(* IEC 61131-3 sources: Dev/Dev_V200/200 (part 10) *)

      iov : ARRAY[0.._Nh_CFG] OF FILT_LIST := [    // v hlavicke je RIADOK a v STLPCOCH su DEV, ktore ho mozu spustat (budu v prowse pre vyber)
            (),     	//  0 Empty
            (),    	//  1 Rmpty Rom
            (),    	//  2 Empty Cat
            (),    	//  3 Empty Zon
//                 0         5         10        15        20        25        30        35	      40        45	     50        55	       60        65
            (n := [0,0,0,0,0,0,0,0,0,0,0,0,0,1,1,1,0,0,0,0,0,0,0,0,0,0,0,0,0,0,0,0,0,0,0,0,0,0,0,0,1,0,0,0,0,0,0,0,0,0,1,0,0,0,0,0,0,0,0,0,0,0,0,0,0,0]) ,    //  4 scn  sceny
            (n := [0,0,0,0,0,0,0,0,0,0,0,0,0,1,1,1,0,0,0,0,0,0,0,0,1,0,0,0,0,0,0,0,0,0,0,0,0,0,0,0,1,0,0,0,0,0,0,0,0,0,1,0,0,0,0,0,0,0,0,0,0,0,0,0,0,0]) ,    //  5 act  akcie
            (n := [0,0,0,0,0,0,0,0,0,0,1,1,1,1,1,0,0,0,0,0,0,0,0,0,0,0,0,0,0,0,0,0,0,0,0,0,0,0,0,0,1,0,0,1,1,0,0,0,0,0,0,0,0,0,0,0,0,0,0,0,0,0,0,0,0,0]) ,    //  6 het  modul kurenia
            (n := [0,0,0,0,0,0,0,0,0,0,0,0,0,0,0,0,0,0,0,0,0,0,0,0,0,0,0,0,0,0,0,0,0,0,0,0,0,0,0,0,0,0,0,0,0,0,0,0,0,0,0,0,0,0,0,0,0,0,0,0,0,0,0,0,0,0]) ,    //  7 kot  kotol
            (n := [0,0,0,0,0,0,0,0,0,0,0,0,0,0,0,0,0,0,0,0,0,0,0,0,0,0,0,0,0,0,0,0,0,0,0,0,0,0,0,0,0,0,0,0,0,0,0,0,0,0,0,0,0,0,0,0,0,0,0,0,0,0,0,0,0,0]) ,    //  8 TVE  termoventil,spirala
            (n := [0,0,0,0,0,0,0,0,0,0,0,0,0,0,0,0,0,0,0,0,0,0,0,0,0,0,0,0,0,0,0,0,0,0,0,0,0,0,0,0,0,0,0,0,0,0,0,0,0,0,0,0,0,0,0,0,0,0,0,0,0,0,0,0,0,0]) ,    //  9 CER  obehove cerpadlo
            (n := [0,0,0,0,0,0,0,0,0,0,0,0,0,1,1,1,0,0,0,0,0,0,0,0,0,0,0,0,0,0,0,0,0,0,0,0,0,0,0,0,1,0,0,0,0,0,0,1,0,0,1,0,0,0,0,0,0,0,0,1,0,0,0,0,0,0]) ,    // 10 SVD  svetlo digital
            (n := [0,0,0,0,0,0,0,0,0,0,0,0,0,1,1,1,0,0,0,0,0,0,0,0,0,0,0,0,0,0,0,0,0,0,0,0,0,0,0,0,1,0,0,0,0,0,0,1,0,0,1,0,0,0,0,0,0,0,0,1,0,0,0,0,0,0]) ,    // 11 SVA  svetlo stivatelne
            (n := [0,0,0,0,0,0,0,0,0,0,0,0,0,1,1,1,0,0,0,0,0,0,0,0,0,0,0,0,0,0,0,0,0,0,0,0,0,0,0,0,1,0,0,0,0,0,0,1,0,0,1,0,0,0,0,0,0,0,0,1,0,0,0,0,0,0]) ,    // 12 RGB  svetlo farebne
//                 0         5         10        15        20        25        30        35	      40        45	     50        55	       60        65
            (n := [0,0,0,0,1,1,1,0,0,0,1,1,1,0,0,0,0,0,0,0,0,1,0,0,0,0,0,0,0,0,1,1,1,0,0,1,0,1,0,0,0,0,1,1,1,0,0,1,0,0,0,0,0,0,0,0,0,0,0,1,0,0,0,0,0,0]) ,    // 13 WSB  ovladac WSB
            (n := [0,0,0,0,1,1,1,0,0,0,1,1,1,0,0,0,0,0,0,0,0,1,0,0,0,0,0,0,0,0,1,1,1,0,0,1,0,1,0,0,0,0,1,1,1,0,0,1,0,0,0,0,0,0,0,0,0,0,0,1,0,0,0,0,0,0]) ,    // 14 TLA  tlacitka
            (n := [0,0,0,0,1,1,1,0,0,0,1,1,1,0,0,0,0,0,0,0,0,1,0,0,0,0,0,0,0,0,0,0,1,0,0,1,0,0,0,0,0,0,0,1,1,0,0,1,0,1,1,0,0,0,0,0,0,0,0,0,0,0,0,0,0,0]) ,    // 15 pir
            (n := [0,0,0,0,0,0,1,0,0,0,0,0,0,0,0,0,0,0,0,0,0,0,0,0,0,0,0,0,0,0,0,0,0,0,0,0,0,0,0,0,0,0,0,0,0,0,0,0,0,1,0,0,0,0,0,0,0,0,0,0,0,0,0,0,0,0]) ,    // 16 teR  teplota-miestnost
            (n := [0,0,0,0,0,0,0,0,0,0,0,0,0,0,0,0,0,0,0,0,0,0,0,0,0,0,0,0,0,0,0,0,0,0,0,0,0,0,0,0,0,0,0,0,0,0,0,0,0,1,0,0,0,0,0,0,0,0,0,0,0,0,0,0,0,0]) ,    // 17 teH  teplota-teleso
            (n := [0,0,0,0,0,0,0,0,0,0,0,0,0,0,0,0,0,0,0,0,0,0,0,0,0,0,0,0,0,0,0,0,0,0,0,0,0,0,0,0,0,0,0,0,0,0,0,0,0,0,0,0,0,0,0,0,0,0,0,0,0,0,0,0,0,0]) ,    // 18 teK  teplota-kotol
            (n := [0,0,0,0,0,0,0,0,0,0,0,0,0,0,0,0,0,0,0,0,0,0,0,0,0,0,0,0,0,0,0,0,0,0,0,0,0,0,0,0,0,0,0,0,0,0,0,0,0,0,0,0,0,0,0,0,0,0,0,0,0,0,0,0,0,0]) ,    // 19 lux  intenzita osvetlenia
            (n := [0,0,0,0,0,0,0,0,0,0,0,0,0,0,0,0,0,0,0,0,0,0,0,0,0,0,0,0,0,0,0,0,0,0,0,0,0,0,0,0,0,0,0,0,0,0,0,0,0,1,0,0,0,0,0,0,0,0,0,0,0,0,0,0,0,0]),     // 20 FAV
            (n := [0,0,0,0,0,0,0,0,0,0,0,0,0,1,1,1,0,0,0,0,0,0,0,0,0,0,0,0,0,0,0,0,0,0,0,1,0,0,0,0,1,0,0,0,0,0,0,1,0,0,1,0,0,0,0,0,0,0,0,1,0,0,0,0,0,0]),     // 21 ZAS  spotrebice
            (n := [0,0,0,0,0,0,0,0,0,0,0,0,0,0,0,0,0,0,0,0,0,0,0,0,0,0,0,0,0,0,0,0,0,0,0,0,0,0,0,0,0,0,0,0,0,0,0,0,0,1,0,0,0,0,0,0,0,0,0,0,0,0,0,0,0,0]),     // 22 USR  uzivatelia
//                 0         5         10        15        20        25        30        35	      40        45	     50        55	       60        65
            (n := [0,0,0,0,0,0,0,0,0,0,0,0,0,0,0,0,0,0,0,0,0,0,0,0,0,0,0,0,0,0,0,0,0,0,0,0,0,0,0,0,0,0,0,0,0,0,0,0,0,0,0,0,0,0,0,0,0,0,0,0,0,0,0,0,0,0]),     // 23 VEN/REK-uperacia
            (n := [0,0,0,0,0,0,0,0,0,0,0,0,0,0,0,0,0,0,0,0,0,0,0,0,0,0,0,0,0,0,0,0,0,0,0,0,0,0,0,0,0,0,0,0,0,0,0,0,0,1,0,0,0,0,0,0,0,0,0,0,0,0,0,0,0,0]),     // 24 KEY
            (n := [0,0,0,0,0,0,0,0,0,0,0,0,0,0,0,0,0,0,0,0,0,0,0,0,0,0,0,0,0,0,0,0,0,0,0,0,0,0,0,0,0,0,0,0,0,0,0,0,0,1,0,0,0,0,0,0,0,0,0,0,0,0,0,0,0,0]),     // 25 RZV - casovy rozvrh PO-NE
            (n := [0,0,0,0,0,0,0,0,0,0,0,0,0,0,0,0,0,0,0,0,0,0,0,0,0,0,0,0,0,0,0,0,0,0,0,0,0,0,0,0,0,0,0,0,0,0,0,0,0,1,0,0,0,0,0,0,0,0,0,0,0,0,0,0,0,0]),     // 26 POI - slider
            (n := [0,0,0,0,0,0,0,0,0,0,0,0,0,0,0,0,0,0,0,0,0,0,0,0,0,0,0,0,0,0,0,0,0,0,0,0,0,0,0,0,0,0,0,0,0,0,0,0,0,1,0,0,0,0,0,0,0,0,0,0,0,0,0,0,0,0]),     // 27 H2O
            (n := [0,0,0,0,0,0,0,0,0,0,0,0,0,0,0,0,0,0,0,0,0,0,0,0,0,0,0,0,0,0,0,0,0,0,0,0,0,0,0,0,0,0,0,0,0,0,0,0,0,1,0,0,0,0,0,0,0,0,0,0,0,0,0,0,0,0]),     // 28 FIRe - len ON/OFF : poziar,dym,CO,CO2,butan...
            (n := [0,0,0,0,0,0,0,0,0,0,0,0,0,0,0,0,0,0,0,0,0,0,0,0,0,0,0,0,0,0,0,0,0,0,0,0,0,0,0,0,0,0,0,0,0,0,0,0,0,1,0,0,0,0,0,0,0,0,0,0,0,0,0,0,0,0]),     // 29 GAS // intenzita (real) CO,CO2,metan,butan,RH
            (n := [0,0,0,0,0,0,0,0,0,0,0,0,0,1,1,0,0,0,0,0,0,0,0,0,0,0,0,0,0,0,0,0,0,0,0,0,0,0,0,0,1,0,0,0,0,0,0,0,0,0,0,0,0,0,0,0,0,0,0,1,0,0,0,0,0,0]),     // 30 MAR garaz,brana,branicka
            (n := [0,0,0,0,0,0,0,0,0,0,0,0,0,1,1,0,0,0,0,0,0,0,0,0,0,0,0,0,0,0,0,0,0,0,0,0,0,0,0,0,1,0,0,0,0,0,0,0,0,0,1,0,0,0,0,0,0,0,0,1,0,0,0,0,0,0]),     // 31 ROL rolety
            (n := [0,0,0,0,0,0,0,0,0,0,0,0,0,1,1,1,0,0,0,0,0,0,0,0,0,0,0,0,0,0,0,0,0,0,0,1,0,0,0,0,1,0,0,0,0,0,0,0,0,0,1,0,0,0,0,0,0,0,0,1,0,0,0,0,0,0]),     // 32 SIR sirena,stroboskop,zvoncek
            (n := [0,0,0,0,0,0,0,0,0,0,0,0,0,0,0,0,0,0,0,0,0,0,0,0,0,0,0,0,0,0,0,0,0,0,0,0,0,0,0,0,0,0,0,0,0,0,0,0,0,1,0,0,0,0,0,0,0,0,0,0,0,0,0,0,0,0]),     // 33 DOR
            (n := [0,0,0,0,0,0,0,0,0,0,0,0,0,0,0,0,0,0,0,0,0,0,0,0,0,0,0,0,0,0,0,0,0,0,0,0,0,0,0,0,0,0,0,0,0,0,0,0,0,1,0,0,0,0,0,0,0,0,0,0,0,0,0,0,0,0]),     // 34 WIN
//                 0         5         10        15        20        25        30        35	      40        45	     50        55	       60        65
            (n := [0,0,0,1,0,0,0,0,0,0,0,0,0,1,1,1,0,0,0,0,0,0,0,0,0,0,0,1,0,0,0,0,0,1,1,0,0,0,0,0,1,0,0,0,0,0,0,0,0,0,1,0,0,0,0,0,0,0,0,0,0,0,0,0,0,0]),     // 35 BLK
            (n := [0,0,0,0,0,0,0,0,0,0,0,0,0,0,0,0,0,0,0,0,0,0,0,0,0,0,0,0,0,0,0,0,0,0,0,0,0,0,0,0,0,0,0,0,0,0,0,0,0,1,0,0,0,0,0,0,0,0,0,0,0,0,0,0,0,0]),     // 36    XXX*BLx
            (n := [0,0,0,0,0,0,0,0,0,0,0,0,0,1,1,0,0,0,0,0,0,0,0,0,0,0,0,0,0,0,0,0,0,0,0,0,0,0,0,0,1,0,0,0,0,0,0,0,0,0,1,0,0,0,0,0,0,0,0,0,0,0,0,0,0,0]),     // 37 BRA,GAR....
            (n := [0,0,0,0,0,0,0,0,0,0,0,0,0,0,0,0,0,0,0,0,0,0,0,0,0,0,0,0,0,0,0,0,0,0,0,0,0,0,0,0,0,0,0,0,0,0,0,0,0,0,0,0,0,0,0,0,0,0,0,0,0,0,0,0,0,0]),     // 38 RFI
            (n := [0,0,0,0,0,0,0,0,0,0,0,0,0,0,0,0,0,0,0,0,0,0,0,0,0,0,0,0,0,0,0,0,0,0,0,0,0,0,0,0,0,0,0,0,0,0,0,0,0,0,0,0,0,0,0,0,0,0,0,0,0,0,0,0,0,0]),     // 39 RFK

            (n := [0,0,0,0,1,1,1,0,0,0,1,1,1,0,0,0,0,0,0,0,0,1,0,0,0,0,0,0,0,0,1,1,1,0,0,1,0,1,0,0,0,0,1,1,1,0,0,1,0,0,0,0,0,0,0,0,0,0,0,1,0,0,0,0,0,0]),     // 40 TGL
            (n := [0,0,0,0,1,1,0,0,0,0,0,0,0,0,0,0,0,0,0,0,0,0,0,0,0,0,0,0,0,0,0,0,0,0,0,0,0,0,0,0,0,0,0,0,0,0,0,0,0,0,0,0,0,0,0,0,0,0,0,0,0,0,0,0,0,0]),     // 41 COX
            (n := [0,0,0,0,1,1,0,0,0,0,0,0,0,0,0,0,0,0,0,0,0,0,0,0,0,0,0,0,0,0,0,0,0,0,0,0,0,0,0,0,0,0,0,0,0,0,0,0,0,1,0,0,0,0,0,0,0,0,0,0,0,0,0,0,0,0]),     // 42 DALI*M
            (n := [0,0,0,0,0,0,0,0,0,0,0,0,0,1,1,1,0,0,0,0,0,0,0,0,0,0,0,0,0,0,0,0,0,0,0,1,0,0,0,0,1,0,0,0,0,0,0,1,0,0,0,0,0,0,0,0,0,0,0,0,0,0,0,0,0,0]),     // 43 DALI - S
            (n := [0,0,0,0,0,0,0,0,0,0,0,0,0,1,1,1,0,0,0,0,0,0,0,0,0,0,0,0,0,0,0,0,0,0,0,1,0,0,0,0,1,0,0,0,0,0,0,1,0,0,0,0,0,0,0,0,0,0,0,0,0,0,0,0,0,0]),     // 44 DALI - GRP
            (n := [0,0,0,0,1,1,0,0,0,0,0,0,0,0,0,0,0,0,0,0,0,0,0,0,0,0,0,0,0,0,0,0,0,0,0,0,0,0,0,0,0,0,0,0,0,0,0,0,0,1,0,0,0,0,0,0,0,0,0,0,0,0,0,0,0,0]),     // 45 SMW - smart way
//                 0         5         10        15        20        25        30        35	      40        45	     50        55	       60        65
            (n := [0,0,0,0,0,0,0,0,0,0,0,0,0,1,0,0,0,0,0,0,0,0,0,0,0,0,0,0,0,0,0,0,0,0,0,0,0,0,0,0,1,0,0,0,0,0,0,0,0,0,0,0,0,0,0,0,0,0,0,0,0,0,0,0,0,0]),     // 46 MSG
            (n := [0,0,0,0,0,0,0,0,0,0,1,1,1,1,1,1,0,0,0,0,0,0,0,0,0,0,0,0,0,0,0,0,0,1,1,0,0,0,0,0,1,0,0,1,0,0,0,0,0,0,0,0,0,0,0,0,0,0,0,0,0,0,0,0,0,0]),     // 47 HEV {HET=rekuperacia}
            (n := [0,0,0,0,0,0,0,0,0,0,0,0,0,0,0,0,0,0,0,0,0,0,0,0,0,0,0,0,0,0,0,0,0,0,0,0,0,0,0,0,0,0,0,0,0,0,0,0,0,0,0,0,0,0,0,0,0,0,0,0,0,0,0,0,0,0]),     // 48 ALA {akcia alarmu}
            (n := [0,0,0,0,0,0,0,0,0,0,0,0,0,1,1,0,0,0,0,0,0,0,0,0,0,0,0,0,0,0,0,0,0,0,0,0,0,0,0,0,1,0,0,0,0,0,0,0,0,0,0,0,0,0,0,0,0,0,0,0,0,0,0,0,0,0]),     // 49 VVO
            (n := [0,0,0,0,1,1,0,0,0,0,1,1,1,0,0,0,0,0,0,0,0,1,0,0,0,0,0,0,0,0,1,1,1,0,0,0,0,0,0,0,0,0,1,1,1,0,0,0,0,1,0,0,0,0,0,0,0,0,0,0,0,0,0,0,0,0])      // 50 TIM
         ];

      in : ARRAY[0.._Nh_CFG] OF FILT_LIST := [ // riadok sa spyta, ci je IN oproti DEV v hlavicke=STLPEC
//                 0         5         10        15        20        25        30        35	      40        45	     50        55	       60        65
            (n := [0,0,0,0,0,0,0,0,0,0,0,0,0,0,0,0,0,0,0,0,0,0,0,0,0,0,0,0,0,0,0,0,0,0,0,0,0,0,0,0,0,0,0,0,0,0,0,0,0,0,0,0,0,0,0,0,0,0,0,0,1,0,0,0,0,0]) ,    //  0  ken pre zachytenie chyby, ked sa odkazuje cf=0
            (n := [0,0,0,1,0,0,1,0,0,0,0,0,0,0,0,0,0,0,0,0,0,0,0,0,0,0,0,0,0,0,0,0,0,0,0,0,0,0,0,0,0,0,0,0,0,0,0,0,0,0,0,0,0,0,0,0,0,0,0,0,1,0,0,0,0,0]) ,    //  1 rom  miestnosti
            (n := [0,0,0,0,1,1,1,1,1,1,1,1,1,1,1,1,1,1,1,1,1,1,1,1,1,1,1,1,1,1,1,1,1,1,1,1,1,1,1,1,1,1,1,1,1,1,1,1,1,1,0,0,0,0,0,0,0,0,0,0,1,0,0,0,0,0]) ,    //  2 cat  kategorie
            (n := [0,1,0,0,0,1,0,0,0,0,0,0,0,0,0,0,0,0,0,0,0,0,0,0,0,0,0,0,0,0,0,0,0,0,0,1,0,0,0,0,0,0,0,0,0,0,0,0,0,0,0,0,0,0,0,0,0,0,0,0,0,0,0,0,0,0]) ,    //  3 zon  zony
            (n := [1,1,1,1,1,0,1,1,1,1,1,1,1,0,0,0,1,1,1,1,1,1,1,1,1,1,1,1,1,1,1,1,1,1,1,0,1,1,1,1,0,1,1,1,1,0,0,0,0,0,0,0,0,0,0,0,0,0,0,0,0,0,0,0,0,0]) ,    //  4 scn  sceny
            (n := [0,0,0,0,0,0,1,1,1,1,1,1,1,0,0,0,1,1,1,1,1,1,1,1,1,1,1,1,1,1,1,1,1,1,1,0,1,1,1,1,0,1,1,1,1,0,0,0,0,1,0,0,0,0,0,0,0,0,0,0,0,0,0,0,0,0]) ,    //  5 act  akcie
            (n := [0,0,0,0,0,0,0,0,0,0,0,0,0,0,0,0,0,0,0,0,0,0,0,0,0,0,0,0,0,0,0,0,0,0,0,0,0,0,0,0,0,0,0,0,0,0,0,0,0,0,0,0,0,0,0,0,0,0,0,0,0,0,0,0,0,0]) ,    //  6 het  modul kurenia
            (n := [0,0,0,0,0,0,1,0,0,0,0,0,0,0,0,0,0,0,0,0,0,0,0,0,0,0,0,0,0,0,0,0,0,0,0,0,0,0,0,0,0,0,0,0,0,0,0,0,0,1,0,0,0,0,0,0,0,0,0,0,0,0,0,0,0,0]) ,    //  7 kot  kotol
            (n := [0,0,0,0,0,0,1,0,0,0,0,0,0,0,0,0,0,1,0,0,0,0,0,0,0,0,0,0,0,0,0,0,0,0,0,0,0,0,0,0,0,0,0,0,0,0,0,0,0,1,0,0,0,0,0,0,0,0,0,0,0,0,0,0,0,0]) ,    //  8 tve  termoventil,spirala
            (n := [0,0,0,0,0,0,1,0,0,0,0,0,0,0,0,0,0,0,0,0,0,0,0,0,0,0,0,0,0,0,0,0,0,0,0,0,0,0,0,0,0,0,0,0,0,0,0,0,0,1,0,0,0,0,0,0,0,0,0,0,0,0,0,0,0,0]) ,    //  9 cer  obehove cerpadlo
            (n := [0,0,0,0,0,0,1,0,0,0,0,0,0,0,0,0,0,0,0,0,0,0,0,0,0,0,0,0,0,0,0,0,0,0,0,0,0,0,0,0,0,0,0,0,0,0,0,1,0,0,0,0,0,0,0,0,0,0,0,0,0,0,0,0,0,0]) ,    // 10 svd  svetlo digital
            (n := [0,0,0,0,0,0,1,0,0,0,0,0,0,0,0,0,0,0,0,0,0,0,0,0,0,0,0,0,0,0,0,0,0,0,0,0,0,0,0,0,0,0,0,0,0,0,0,1,0,0,0,0,0,0,0,0,0,0,0,0,0,0,0,0,0,0]) ,    // 11 sva  svetlo stievatelne
            (n := [0,0,0,0,0,0,1,0,0,0,0,0,0,0,0,0,0,0,0,0,0,0,0,0,0,0,0,0,0,0,0,0,0,0,0,0,0,0,0,0,0,0,0,0,0,0,0,1,0,0,0,0,0,0,0,0,0,0,0,0,0,0,0,0,0,0]) ,    // 12 rgb  svetlo farebne
            (n := [1,1,1,1,1,1,1,1,1,1,1,1,1,1,1,1,1,1,1,1,1,1,1,1,1,1,1,1,1,1,1,1,1,1,1,1,1,1,1,1,1,1,1,1,1,1,1,1,1,1,1,1,1,1,1,1,1,1,1,1,1,1,1,1,1,1]) ,    // 13 wsb  ovladac WSB
            (n := [1,1,1,1,1,1,1,1,1,1,1,1,1,1,1,1,1,1,1,1,1,1,1,1,1,1,1,1,1,1,1,1,1,1,1,1,1,1,1,1,1,1,1,1,1,1,1,1,1,1,1,1,1,1,1,1,1,1,1,1,1,1,1,1,1,1]) ,    // 14 tla  tlacitka
            (n := [1,1,1,1,1,1,1,1,1,1,1,1,1,1,1,1,1,1,1,1,1,1,1,1,1,1,1,1,1,1,1,1,1,1,1,1,1,1,1,1,1,1,1,1,1,1,1,1,1,1,1,1,1,1,1,1,1,1,1,1,1,1,1,1,1,1]) ,    // 15 pir
            (n := [0,1,1,1,1,1,1,1,1,1,1,1,1,1,1,1,1,1,1,1,1,1,1,1,1,1,1,1,1,1,1,1,1,1,1,1,1,1,1,1,1,1,1,1,1,1,1,1,1,1,1,1,1,1,1,1,1,1,1,1,1,1,1,1,1,1]) ,    // 16 teR  teplota miestnost
            (n := [0,1,1,1,1,1,1,1,1,1,1,1,1,1,1,1,1,1,1,1,1,1,1,1,1,1,1,1,1,1,1,1,1,1,1,1,1,1,1,1,1,1,1,1,1,1,1,1,1,1,1,1,1,1,1,1,1,1,1,1,1,1,1,1,1,1]) ,    // 17 teH  teplot radiator
            (n := [0,1,1,1,1,1,1,1,1,1,1,1,1,1,1,1,1,1,1,1,1,1,1,1,1,1,1,1,1,1,1,1,1,1,1,1,1,1,1,1,1,1,1,1,1,1,1,1,1,1,1,1,1,1,1,1,1,1,1,1,1,1,1,1,1,1]) ,    // 18 teK  teplota kotol
//                 0         5         10        15        20        25        30        35	      40        45	     50        55	       60        65
            (n := [0,1,1,1,1,1,1,1,1,1,1,1,1,1,1,1,1,1,1,1,1,1,1,1,1,1,1,1,1,1,1,1,1,1,1,1,1,1,1,1,1,1,1,1,1,1,1,1,1,0,1,0,0,0,0,0,0,0,0,0,1,0,0,0,0,0]) ,    // 19 lux  intenzita osvetlenia
            (n := [0,0,0,0,1,1,0,0,0,0,0,0,0,0,0,0,0,0,0,0,0,0,0,0,0,0,0,0,0,0,0,0,0,0,0,0,0,0,0,0,0,0,0,0,0,0,0,0,0,0,0,0,0,0,0,0,0,0,0,0,0,0,0,0,0,0]) ,    // 20 FAV
            (n := [0,0,0,0,0,0,0,0,0,0,0,0,0,0,0,0,0,0,0,0,0,0,0,0,0,0,0,0,0,0,0,0,0,0,0,0,0,0,0,0,0,0,0,0,0,0,0,0,0,0,0,0,0,0,0,0,0,0,0,0,0,0,0,0,0,0]) ,    // 21 ZAS  spotrebice
            (n := [0,0,0,0,1,1,0,0,0,0,0,0,0,0,0,0,0,0,0,0,0,0,0,0,0,0,0,0,0,0,0,0,0,0,0,0,0,0,0,0,0,0,0,0,0,0,0,0,0,0,0,0,0,0,0,0,0,0,0,0,0,0,0,0,0,0]) ,    // 22 Usr  uzivatelia

            (n := [0,0,0,0,0,0,0,0,0,0,0,0,0,0,0,0,0,0,0,0,0,0,0,0,0,0,0,0,0,0,0,0,0,0,0,0,0,0,0,0,0,0,0,0,0,0,0,0,0,0,0,0,0,0,0,0,0,0,0,0,0,0,0,0,0,0]) ,    // 23 VEN
            (n := [1,1,1,1,1,1,1,1,1,1,1,1,1,1,1,1,1,1,1,1,1,1,1,1,1,1,1,1,1,1,1,1,1,1,1,1,1,1,1,1,1,1,1,1,1,1,1,1,1,1,1,1,1,1,1,1,1,1,1,1,1,1,1,1,1,1]),     // 24 KEY
            (n := [1,1,1,1,1,1,1,1,1,1,1,1,1,1,1,1,1,1,1,1,1,1,1,1,1,1,1,1,1,1,1,1,1,1,1,1,1,1,1,1,1,1,1,1,1,1,1,1,1,1,1,0,0,0,0,0,0,0,0,0,1,0,0,0,0,0]),     // 25 PRG - casovy program
            (n := [0,0,0,0,0,0,0,0,0,0,0,0,0,0,0,0,0,0,0,0,0,0,0,0,0,0,0,0,0,0,0,0,0,0,0,0,0,0,0,0,0,0,0,0,0,0,0,0,0,1,0,0,0,0,0,0,0,0,0,0,0,0,0,0,0,0]),     // 26 Stykace - okruhy
            (n := [1,1,1,1,1,1,1,1,1,1,1,1,1,1,1,1,1,1,1,1,1,1,1,1,1,1,1,1,1,1,1,1,1,1,1,1,1,1,1,1,1,1,1,1,1,1,1,1,1,1,1,1,1,1,1,1,1,1,1,1,1,1,1,1,1,1]),     // 27 H2O
            (n := [1,1,1,1,1,1,1,1,1,1,1,1,1,1,1,1,1,1,1,1,1,1,1,1,1,1,1,1,1,1,1,1,1,1,1,1,1,1,1,1,1,1,1,1,1,1,1,1,1,1,1,1,1,1,1,1,1,1,1,1,1,1,1,1,1,1]),     // 28 FIRe - len ON/OFF : poziar,dym,CO,CO2,butan...
            (n := [1,1,1,1,1,1,1,1,1,1,1,1,1,1,1,1,1,1,1,1,1,1,1,1,1,1,1,1,1,1,1,1,1,1,1,1,1,1,1,1,1,1,1,1,1,1,1,1,1,1,1,1,1,1,1,1,1,1,1,1,1,1,1,1,1,1]),     // 29 GAS // intenzita (real) CO,CO2,metan,butan,RH
            (n := [0,0,0,0,0,0,0,0,0,0,0,0,0,0,0,0,0,0,0,0,0,0,0,0,0,0,0,0,0,0,0,0,0,0,0,0,0,0,0,0,0,0,0,0,0,0,0,0,0,1,0,0,0,0,0,0,0,0,0,0,0,0,0,0,0,0]),     // 30 MAR
            (n := [0,0,0,0,0,0,0,0,0,0,0,0,0,0,0,0,0,0,0,0,0,0,0,0,0,0,0,0,0,0,0,0,0,0,0,0,0,0,0,0,0,0,0,0,0,0,0,0,0,1,0,0,0,0,0,0,0,0,0,0,0,0,0,0,0,0]),     // 31 ROL rolety
            (n := [0,0,0,0,0,0,0,0,0,0,0,0,0,0,0,0,0,0,0,0,0,0,0,0,0,0,0,0,0,0,0,0,0,0,0,0,0,0,0,0,0,0,0,0,0,0,0,0,0,1,0,0,0,0,0,0,0,0,0,0,0,0,0,0,0,0]),     // 32 SIR sirena,stroboskop,zvoncek
            (n := [1,1,1,1,1,1,1,1,1,1,1,1,1,1,1,1,1,1,1,1,1,1,1,1,1,1,1,1,1,1,1,1,1,1,1,1,1,1,1,1,1,1,1,1,1,1,1,1,1,1,1,1,1,1,1,1,1,1,1,1,1,1,1,1,1,1]),     // 32 DOR
            (n := [1,1,1,1,1,1,1,1,1,1,1,1,1,1,1,1,1,1,1,1,1,1,1,1,1,1,1,1,1,1,1,1,1,1,1,1,1,1,1,1,1,1,1,1,1,1,1,1,1,1,1,1,1,1,1,1,1,1,1,1,1,1,1,1,1,1]),     // 34 WIN
            (n := [0,0,0,1,1,1,0,0,0,0,1,1,1,0,0,0,0,0,0,0,0,1,0,1,0,0,0,0,0,0,0,1,1,0,0,0,0,1,0,0,0,0,0,0,0,0,0,0,0,1,0,0,0,0,0,0,0,0,0,0,0,0,0,0,0,0]),     // 35 BLK
            (n := [0,0,0,0,0,0,0,0,0,0,0,0,0,0,0,0,0,0,0,0,0,0,0,0,0,0,0,0,0,0,0,0,0,0,0,0,0,0,0,0,0,0,0,0,0,0,0,0,0,1,0,0,0,0,0,0,0,0,0,0,0,0,0,0,0,0]),     // 36 XXX
            (n := [0,0,0,0,0,0,0,0,0,0,0,0,0,0,0,0,0,0,0,0,0,0,0,0,0,0,0,0,0,0,0,0,0,0,0,0,0,0,0,0,0,0,0,0,0,0,0,0,0,1,0,0,0,0,0,0,0,0,0,0,0,0,0,0,0,0]),     // 37 BRA
            (n := [0,0,0,0,1,1,0,0,0,0,0,0,0,0,0,0,0,0,0,0,0,0,0,0,0,0,0,0,0,0,0,0,0,0,0,0,0,0,0,0,0,0,0,0,0,0,0,0,0,1,0,0,0,0,0,0,0,0,0,0,0,0,0,0,0,0]),     // 38 RFI
            (n := [0,0,0,0,1,1,0,0,0,0,0,0,0,0,0,0,0,0,0,0,0,0,0,0,0,0,0,0,0,0,0,0,0,0,0,0,0,0,0,0,0,0,0,0,0,0,0,0,0,1,0,0,0,0,0,0,0,0,0,0,0,0,0,0,0,0]),     // 39 RFK
//                 0         5         10        15        20        25        30        35	      40        45	     50        55	       60        65
            (n := [1,1,1,1,1,1,1,1,1,1,1,1,1,1,1,1,1,1,1,1,1,1,1,1,1,1,1,1,1,1,1,1,1,1,1,1,1,1,1,1,1,1,1,1,1,1,1,1,1,1,1,1,1,1,1,1,1,1,1,1,1,1,1,1,1,1]),     // 40 TGL
            (n := [0,0,0,0,1,1,0,0,0,0,0,0,0,0,0,0,0,0,0,0,0,0,0,0,0,0,0,0,0,0,0,0,0,0,0,0,0,0,0,0,0,0,0,0,0,0,0,1,0,0,0,0,0,0,0,0,0,0,0,0,0,0,0,0,0,0]),     // 41 BTN
            (n := [0,0,0,0,0,0,0,0,0,0,0,0,0,0,0,0,0,0,0,0,0,0,0,0,0,0,0,0,0,0,0,0,0,0,0,0,0,0,0,0,0,0,0,0,0,0,0,1,0,0,0,0,0,0,0,0,0,0,0,0,0,0,0,0,0,0]),     // 42 DL-ma
            (n := [0,0,0,0,0,0,0,0,0,0,0,0,0,0,0,0,0,0,0,0,0,0,0,0,0,0,0,0,0,0,0,0,0,0,0,0,0,0,0,0,0,0,0,0,0,0,0,1,0,0,0,0,0,0,0,0,0,0,0,0,0,0,0,0,0,0]),     // 43 DL-slave
            (n := [0,0,0,0,0,0,0,0,0,0,0,0,0,0,0,0,0,0,0,0,0,0,0,0,0,0,0,0,0,0,0,0,0,0,0,0,0,0,0,0,0,0,0,0,0,0,0,1,0,0,0,0,0,0,0,0,0,0,0,0,0,0,0,0,0,0]),     // 44 DL-group
            (n := [0,0,0,0,1,1,0,0,0,0,0,0,0,0,0,0,0,0,0,0,0,0,0,0,0,0,0,0,0,0,0,0,0,0,0,0,0,0,0,0,0,0,0,0,0,0,0,1,0,0,0,0,0,0,0,0,0,0,0,0,0,0,0,0,0,0]),     // 45 SMW
            (n := [0,0,0,0,1,1,0,0,0,0,0,0,0,0,0,0,0,0,0,0,0,0,0,0,0,0,0,0,0,0,0,0,0,0,0,0,0,0,0,0,0,0,0,0,0,0,0,0,0,0,0,0,0,0,0,0,0,0,0,0,0,0,0,0,0,0]),     // 46 MSG
            (n := [0,0,0,0,0,0,0,0,0,0,0,0,0,0,0,0,0,0,0,0,0,0,0,0,0,0,0,0,0,0,0,0,0,0,0,0,0,0,0,0,0,0,0,0,0,0,0,0,0,0,0,0,0,0,0,0,0,0,0,0,0,0,0,0,0,0]),     // 47 HEV
            (n := [0,0,0,0,0,1,0,0,0,0,0,0,0,0,0,0,0,0,0,0,0,0,0,0,0,0,0,0,0,0,0,0,0,0,0,0,0,0,0,0,0,0,0,0,0,0,0,0,0,0,0,0,0,0,0,0,0,0,0,0,0,0,0,0,0,0]),     // 48 ALA
            (n := [0,0,0,0,0,0,0,0,0,0,0,0,1,1,0,0,0,0,0,0,0,0,0,0,0,0,0,0,0,0,0,0,0,0,0,0,0,0,0,0,1,0,0,0,0,0,0,0,0,0,0,0,0,0,0,0,0,0,0,0,0,0,0,0,0,0]),     // 49 VVO
            (n := [1,1,1,1,1,1,1,1,1,1,1,1,1,1,1,1,1,1,1,1,1,1,1,1,1,1,1,1,1,1,1,1,1,1,1,1,1,1,1,1,1,1,1,1,1,1,1,1,1,1,1,1,1,1,1,1,1,1,1,1,1,1,1,1,1,1])      // 50 TIM

				];
   END_STRUCT

   NH_FRM_235   {HIDDEN}     : STRUCT
//      typ : USINT := 235;
      hed : NH_FRM_HED := (Name:='_235',wht:=0) ;
      DevToCat : ARRAY[0.._Nh_CFG] OF FILT_LIST := [   // DEV (v riadku) vstupuje do CAT (stlpec)
			(n := [0,0,0,0,0,0,0,0,0,0,0,0,0,0,0,0,0,0,0,0,0,0,0,0,0,0,0,0,0,0,0,0,0,0,0,0,0,0,0,0,0,0,0,0,0,0,0,0,0,0,0,0,0,0,0,0,0,0,0,0,0,0,0,0,0,0,0,0,0,0,0]),
// 1          	 0         5         10        15        20        25        30        35	      40        45	     50        55	       60        65        70
			(n := [0,0,0,0,0,0,0,0,0,0,0,0,0,0,0,0,0,0,0,0,0,0,0,0,0,0,0,0,0,0,0,0,0,0,0,0,0,0,0,0,0,0,0,0,0,0,0,0,0,0,0,0,0,0,0,0,0,0,0,0,0,0,0,0,0,0,0,0,0,0,0]),	// ROM
			(n := [0,0,0,0,0,0,0,0,0,0,0,0,0,0,0,0,0,0,0,0,0,0,0,0,0,0,0,0,0,0,0,0,0,0,0,0,0,0,0,0,0,0,0,0,0,0,0,0,0,0,0,0,0,0,0,0,0,0,0,0,0,0,0,0,0,0,0,0,0,0,0]),
			(n := [0,0,0,0,0,0,0,0,0,0,0,0,0,0,0,0,0,0,0,0,0,0,0,0,0,0,0,0,0,0,0,0,0,0,0,0,0,0,0,0,0,0,0,0,0,0,0,0,0,0,0,0,0,0,0,0,0,0,0,0,0,0,0,0,0,0,0,0,0,0,0]),  // ZON
			(n := [0,0,0,0,0,0,0,0,0,0,0,0,0,0,0,0,0,0,0,0,0,0,0,0,0,0,0,0,0,0,0,0,0,0,0,0,0,0,0,0,0,0,0,0,0,0,0,0,0,0,0,0,0,1,0,0,0,0,0,0,0,0,0,0,0,0,0,0,0,0,0]),	// SCN
			(n := [0,0,0,0,0,0,0,0,0,0,0,0,0,0,0,0,0,0,0,0,0,0,0,0,0,0,0,0,0,0,0,0,0,0,0,0,0,0,0,0,0,0,0,0,0,0,0,0,0,0,0,0,0,0,0,0,0,0,0,0,0,0,0,0,0,0,0,0,0,0,0]),	// ACT
			(n := [0,0,0,0,0,1,0,0,0,0,0,0,0,0,0,0,0,0,0,0,0,0,0,0,0,0,0,0,0,0,0,0,0,0,0,0,0,0,0,0,0,0,0,0,0,0,0,0,0,0,0,0,0,0,0,0,0,0,0,0,0,0,0,0,0,0,0,0,0,0,0]),  // 6  HET
			(n := [0,0,0,0,0,0,0,0,0,0,0,0,0,0,0,0,0,0,0,0,0,0,0,0,0,0,0,0,0,0,0,0,0,0,0,0,0,0,0,1,0,0,0,0,0,0,0,0,0,0,0,0,0,0,0,0,0,0,0,0,0,0,0,0,0,0,0,0,0,0,0]),	// 7 KOT
			(n := [0,0,0,0,0,0,0,0,0,0,0,0,0,0,0,0,0,0,0,0,0,0,0,0,0,0,0,0,0,0,0,0,0,0,0,0,0,0,0,1,0,0,0,0,0,0,0,0,0,0,0,0,0,0,0,0,0,0,0,0,0,0,0,0,0,0,0,0,0,0,0]),	// 8 TVE
			(n := [0,0,0,0,0,0,0,0,0,0,0,0,0,0,0,0,0,0,0,0,0,0,0,0,0,0,0,0,0,0,0,0,0,0,0,0,0,0,0,1,0,0,0,0,0,0,0,0,0,0,0,0,0,0,0,0,0,0,0,0,0,0,0,0,0,0,0,0,0,0,0]),  // 9 CER
			(n := [0,1,0,0,0,0,0,0,0,0,0,0,0,0,0,0,0,0,0,0,0,0,0,0,0,0,0,0,0,0,0,0,0,0,0,0,0,0,0,0,0,0,0,0,0,0,0,0,0,0,0,0,0,0,0,0,0,0,0,0,0,0,0,0,0,0,0,0,0,0,0]),	//10 SVE
// 11         	 0         5         10        15        20        25        30        35	      40        45	     50        55	       60        65        70
			(n := [0,1,0,0,0,0,0,0,0,0,0,0,0,0,0,0,0,0,0,0,0,0,0,0,0,0,0,0,0,0,0,0,0,0,0,0,0,0,0,0,0,0,0,0,0,0,0,0,0,0,0,0,0,0,0,0,0,0,0,0,0,0,0,0,0,0,0,0,0,0,0]),	// sva
			(n := [0,1,0,0,0,0,0,0,0,0,0,0,0,0,0,0,0,0,0,0,0,0,0,0,0,0,0,0,0,0,0,0,0,0,0,0,0,0,0,0,0,0,0,0,0,0,0,0,0,0,0,0,0,0,0,0,0,0,0,0,0,0,0,0,0,0,0,0,0,0,0]),
			(n := [0,0,0,0,0,0,0,0,0,0,0,0,0,0,0,0,0,0,0,0,0,0,0,0,1,0,0,0,0,0,0,0,0,0,0,0,0,0,0,0,0,0,0,0,0,0,0,0,0,0,0,0,0,0,0,0,0,0,0,0,0,0,0,0,0,0,0,0,0,0,0]),
			(n := [0,0,0,0,0,0,0,0,0,0,0,0,0,0,0,0,0,0,0,0,0,0,0,0,1,0,0,0,0,0,0,0,0,0,0,0,0,0,0,0,0,0,0,0,0,0,0,0,0,0,0,0,0,0,0,0,0,0,0,0,0,0,0,0,0,0,0,0,0,0,0]),	// SVE
			(n := [0,0,0,0,0,0,0,0,0,0,0,0,0,0,0,1,0,0,0,0,0,0,0,0,0,0,0,0,0,0,0,0,0,0,0,0,0,0,0,0,0,0,0,0,0,0,0,0,0,0,0,0,0,0,0,0,0,0,0,0,0,0,0,0,0,0,0,0,0,0,0]),
			(n := [0,0,0,0,0,0,0,0,0,0,0,0,0,0,1,0,0,0,0,0,0,0,0,0,0,0,0,0,0,0,0,0,0,0,0,0,0,0,0,0,0,0,0,0,0,0,0,0,0,0,0,0,0,0,0,0,0,0,0,0,0,0,0,0,0,0,0,0,0,0,0]),  // 16 ter
			(n := [0,0,0,0,0,0,0,0,0,0,0,0,0,0,1,0,0,0,0,0,0,0,0,0,0,0,0,0,0,0,0,0,0,0,0,0,0,0,0,0,0,0,0,0,0,0,0,0,0,0,0,0,0,0,0,0,0,0,0,0,0,0,0,0,0,0,0,0,0,0,0]),	// 17 teh
			(n := [0,0,0,0,0,0,0,0,0,0,0,0,0,0,1,0,0,0,0,0,0,0,0,0,0,0,0,0,0,0,0,0,0,0,0,0,0,0,0,0,0,0,0,0,0,0,0,0,0,0,0,0,0,0,0,0,0,0,0,0,0,0,0,0,0,0,0,0,0,0,0]),	// 18 tek
			(n := [0,0,0,0,0,0,0,0,0,0,0,0,0,0,0,0,1,0,0,0,0,0,0,0,0,0,0,0,0,0,0,0,0,0,0,0,0,0,0,0,0,0,0,0,0,0,0,0,0,0,0,0,0,0,0,0,0,0,0,0,0,0,0,0,0,0,0,0,0,0,0]),  // 18 lux
			(n := [0,0,0,0,0,0,0,0,0,0,0,0,0,0,0,0,0,0,0,0,0,0,0,0,0,0,0,0,0,0,0,0,0,0,0,0,0,0,0,0,0,0,0,0,0,0,0,0,0,0,0,0,0,0,0,0,0,0,0,0,0,0,0,0,0,0,0,0,0,0,0]),	// 20 fav
// 21         	 0         5         10        15        20        25        30        35	      40        45	     50        55	       60        65        70
			(n := [0,0,1,0,0,0,0,0,0,0,0,0,0,0,0,0,0,0,0,0,0,0,0,0,0,0,0,0,0,0,0,0,0,0,0,0,0,0,0,0,0,0,0,0,0,0,0,0,0,0,0,0,0,0,0,0,0,0,0,0,0,0,0,0,0,0,0,0,0,0,0]),	// 21 zas
			(n := [0,0,0,0,0,0,0,0,0,0,0,0,0,0,0,0,0,0,0,0,0,0,0,0,0,0,0,0,0,0,0,1,0,0,0,0,0,0,0,0,0,0,0,0,0,0,0,0,0,0,0,0,0,0,0,0,0,0,0,0,0,0,0,0,0,0,0,0,0,0,0]),	// 22 usr
			(n := [0,0,0,0,0,0,0,0,0,0,0,0,0,0,0,0,0,0,0,0,0,0,0,0,0,0,0,0,0,0,0,0,0,0,0,0,0,0,0,0,0,0,0,0,0,0,0,0,0,0,0,1,0,0,0,0,0,0,0,0,0,0,0,0,0,0,0,0,0,0,0]),  // 23 rek = TVE pre vetranie
			(n := [0,0,0,0,0,0,0,0,0,0,0,0,0,0,0,0,0,0,0,0,0,0,0,0,0,1,0,0,0,0,0,0,0,0,0,0,0,0,0,0,0,0,0,0,0,0,0,0,0,0,0,0,0,0,0,0,0,0,0,0,0,0,0,0,0,0,0,0,0,0,0]),	// 24 key
			(n := [0,0,0,0,0,0,0,0,0,0,0,0,0,0,0,0,0,0,0,0,0,0,0,0,0,0,0,0,0,0,0,0,0,0,0,0,0,0,0,0,0,0,0,0,0,0,0,0,0,0,0,0,0,0,0,0,0,0,0,0,0,0,0,0,0,0,0,0,0,0,0]),
			(n := [0,0,0,0,0,0,0,0,0,0,0,0,0,0,0,0,0,0,0,0,0,0,0,0,0,0,0,0,0,0,0,0,0,0,0,0,0,0,0,0,0,0,0,0,0,0,0,0,0,0,0,0,0,0,0,0,0,0,0,0,0,0,0,0,0,0,0,0,0,0,0]),
			(n := [0,0,0,0,0,0,0,0,0,0,0,0,0,0,0,0,0,0,0,1,0,0,0,0,0,0,0,0,0,0,0,0,0,0,0,0,0,0,0,0,0,0,0,0,0,0,0,0,0,0,0,0,0,0,0,0,0,0,0,0,0,0,0,0,0,0,0,0,0,0,0]),	// SVE
			(n := [0,0,0,0,0,0,0,0,0,0,0,0,0,0,0,0,0,0,0,0,0,0,0,0,0,0,0,0,0,0,0,0,0,0,0,0,0,0,0,0,0,0,0,0,0,0,1,0,0,0,0,0,0,0,0,0,0,0,0,0,0,0,0,0,0,0,0,0,0,0,0]),
			(n := [0,0,0,0,0,0,0,0,0,0,0,0,0,0,0,0,0,0,0,0,0,0,0,0,0,0,0,0,0,0,0,0,0,0,0,0,0,0,0,0,0,0,0,0,0,0,0,0,0,0,1,0,0,0,0,0,0,0,0,0,0,0,0,0,0,0,0,0,0,0,0]),
			(n := [0,0,0,1,0,0,0,0,0,0,0,0,0,0,0,0,0,0,0,0,0,0,0,0,0,0,0,0,0,0,0,0,0,0,0,0,0,0,0,0,0,0,0,0,0,0,0,0,0,0,0,0,0,0,0,0,0,0,0,0,0,0,0,0,0,0,0,0,0,0,0]),	// SVE
// 31         	 0         5         10        15        20        25        30        35	      40        45	     50        55	       60        65        70
			(n := [0,0,0,1,0,0,0,0,0,0,0,0,0,0,0,0,0,0,0,0,0,0,0,0,0,0,0,0,0,0,0,0,0,0,0,0,0,0,0,0,0,0,0,0,0,0,0,0,0,0,0,0,0,0,0,0,0,0,0,0,0,0,0,0,0,0,0,0,0,0,0]),	// SVE
			(n := [0,0,0,0,0,0,1,0,0,0,0,0,0,0,0,0,0,0,0,0,0,0,0,0,0,0,0,0,0,0,0,0,0,0,0,0,0,0,0,0,0,0,0,0,0,0,0,0,0,0,0,0,0,0,0,0,0,0,0,0,0,0,0,0,0,0,0,0,0,0,0]),	// SIR
			(n := [0,0,0,0,0,0,0,0,0,0,0,0,0,0,0,0,0,0,0,0,0,0,0,0,0,0,0,0,0,0,0,0,0,0,0,0,0,0,0,0,0,0,0,0,0,1,0,0,0,0,0,0,0,0,0,0,0,0,0,0,0,0,0,0,0,0,0,0,0,0,0]),  // DOR
			(n := [0,0,0,0,0,0,0,0,0,0,0,0,0,0,0,0,0,0,0,0,0,0,0,0,0,0,0,0,0,0,0,0,0,0,0,0,0,0,0,0,0,0,0,0,1,0,0,0,0,0,0,0,0,0,0,0,0,0,0,0,0,0,0,0,0,0,0,0,0,0,0]),	// WIN
			(n := [0,0,0,0,0,0,0,0,0,0,0,0,0,0,0,0,0,0,0,0,0,0,0,0,0,0,0,0,0,0,0,0,0,0,0,0,0,0,0,0,0,0,0,0,0,0,0,0,0,0,0,0,0,0,0,0,0,0,0,0,0,0,0,0,0,0,0,0,0,0,0]),
			(n := [0,0,0,0,0,0,0,0,0,0,0,0,0,0,0,0,0,0,0,0,0,0,0,0,0,0,0,0,0,0,0,0,0,0,0,0,0,0,0,0,0,0,0,0,0,0,0,0,0,0,0,0,0,0,0,0,0,0,0,0,0,0,0,0,0,0,0,0,0,0,0]),
			(n := [0,0,0,0,0,0,0,1,0,0,0,0,0,0,0,0,0,0,0,0,0,0,0,0,0,0,0,0,0,0,0,0,0,0,0,0,0,0,0,0,0,0,0,0,0,0,0,0,0,0,0,0,0,0,0,0,0,0,0,0,0,0,0,0,0,0,0,0,0,0,0]),	// SVE
			(n := [0,0,0,0,0,0,0,0,0,0,0,0,0,0,0,0,0,0,0,0,0,0,1,0,0,0,0,0,0,0,0,0,0,0,0,0,0,0,0,0,0,0,0,0,0,0,0,0,0,0,0,0,0,0,0,0,0,0,0,0,0,0,0,0,0,0,0,0,0,0,0]),
			(n := [0,0,0,0,0,0,0,0,0,0,0,0,0,0,0,0,0,0,0,0,0,0,0,0,0,0,0,0,0,0,0,0,0,0,0,0,0,1,0,0,0,0,0,0,0,0,0,0,0,0,0,0,0,0,0,0,0,0,0,0,0,0,0,0,0,0,0,0,0,0,0]),
			(n := [0,0,0,0,0,0,0,0,0,0,0,0,0,0,0,0,0,0,0,0,0,0,0,0,1,0,0,0,0,0,0,0,0,0,0,0,0,0,0,0,0,0,0,0,0,0,0,0,0,0,0,0,0,0,0,0,0,0,0,0,0,0,0,0,0,0,0,0,0,0,0]),	// SVE
// 41         	 0         5         10        15        20        25        30        35	      40        45	     50        55	       60        65        70
			(n := [0,0,0,0,0,0,0,0,0,0,0,0,0,0,0,0,0,0,0,0,0,0,0,0,0,0,0,0,0,0,0,0,0,0,0,0,0,0,0,0,0,0,0,1,0,0,0,0,1,0,0,0,0,0,0,0,0,0,0,0,0,0,0,0,0,0,0,0,0,0,0]),	//
			(n := [0,0,0,0,0,0,0,0,0,0,0,0,0,0,0,0,0,0,0,0,0,0,0,0,0,0,0,0,0,0,0,0,0,0,0,1,0,0,0,0,0,0,0,0,0,0,0,0,0,0,0,0,0,0,0,0,0,0,0,0,0,0,0,0,0,0,0,0,0,0,0]),
			(n := [0,1,0,0,0,0,0,0,0,0,0,0,0,0,0,0,0,0,0,0,0,0,0,0,0,0,0,0,0,0,0,0,0,0,0,0,0,0,0,0,0,0,0,0,0,0,0,0,0,0,0,0,0,0,0,0,0,0,0,0,0,0,0,0,0,0,0,0,0,0,0]),
			(n := [0,0,0,0,0,0,0,0,0,0,0,0,0,0,0,0,0,0,0,0,0,0,0,0,0,0,0,0,0,0,0,0,0,0,0,0,0,0,0,0,0,0,0,0,0,0,0,0,0,0,0,0,0,0,1,0,0,0,0,0,0,0,0,0,0,0,0,0,0,0,0]),	// SVE
			(n := [0,0,0,0,0,0,0,0,0,0,0,0,0,0,0,0,0,0,0,0,0,0,0,0,0,0,0,0,0,0,0,0,0,0,0,0,0,0,0,0,0,0,0,0,0,0,0,0,0,0,0,0,0,0,0,0,0,0,0,0,0,0,0,0,0,0,0,0,0,0,0]),
			(n := [0,0,0,0,0,0,0,0,0,0,0,0,0,0,0,0,0,0,0,0,0,0,0,0,0,0,0,0,0,0,0,0,0,0,0,0,0,0,0,0,0,0,0,0,0,0,0,0,0,0,0,0,0,0,0,0,1,1,0,0,0,0,0,0,0,0,0,0,0,0,0]),  // 46 MSG
			(n := [0,0,0,0,1,0,0,0,0,0,0,0,0,0,0,0,0,0,0,0,0,0,0,0,0,0,0,0,0,0,0,0,0,0,0,0,0,0,0,0,0,0,0,0,0,0,0,0,0,0,0,0,0,0,0,0,0,0,0,0,0,0,0,0,0,0,0,0,0,0,0]),	// 47 HEV - regulator vetrania
			(n := [0,0,0,0,0,0,0,0,0,0,0,0,0,0,0,0,0,0,0,0,0,0,0,0,0,0,0,0,0,0,0,0,0,0,0,0,0,0,0,0,0,0,0,0,0,0,0,0,0,0,0,0,0,0,0,1,0,0,0,0,0,0,0,0,0,0,0,0,0,0,0]),	// 48 ALA
			(n := [0,0,0,0,0,0,1,0,0,0,0,0,0,0,0,0,0,0,0,0,0,0,0,0,0,0,0,0,0,0,0,0,0,0,0,0,0,0,0,0,0,0,0,0,0,0,0,0,0,0,0,0,0,0,0,0,0,0,0,0,0,0,0,0,0,0,0,0,0,0,0]),  // VVO
			(n := [0,0,0,0,0,0,0,0,0,0,0,0,0,0,0,0,0,0,0,0,0,0,0,0,0,0,0,0,0,0,0,0,0,0,0,0,0,0,0,0,0,0,0,0,0,0,0,0,0,0,0,0,0,0,0,0,0,0,0,0,0,0,0,0,0,0,0,0,0,0,0]),
// 51         	 0         5         10        15        20        25        30        35	      40        45	     50        55	       60        65        70
			(n := [0,0,0,0,0,0,0,0,0,0,0,0,0,0,0,0,0,0,0,0,0,0,0,0,0,0,0,0,0,0,0,0,0,0,0,0,0,0,0,0,0,0,0,0,0,0,0,0,0,0,0,0,0,0,0,0,0,0,0,0,0,0,0,0,0,0,0,0,0,0,0]),	// SVE
			(n := [0,0,0,0,0,0,0,0,0,0,0,0,0,0,0,0,0,0,0,0,0,0,0,0,0,0,0,0,0,0,0,0,0,0,0,0,0,0,0,0,0,0,0,0,0,0,0,0,0,0,0,0,0,0,0,0,0,0,0,0,0,0,0,0,0,0,0,0,0,0,0]),
			(n := [0,0,0,0,0,0,0,0,0,0,0,0,0,0,0,0,0,0,0,0,0,0,0,0,0,0,0,0,0,0,0,0,0,0,0,0,0,0,0,0,0,0,0,0,0,0,0,0,0,0,0,0,0,0,0,0,0,0,0,0,0,0,0,0,0,0,0,0,0,0,0]),
			(n := [0,0,0,0,0,0,0,0,0,0,0,0,0,0,0,0,0,0,0,0,0,0,0,0,0,0,0,0,0,0,0,0,0,0,0,0,0,0,0,0,0,0,0,0,0,0,0,0,0,0,0,0,0,0,0,0,0,0,0,0,0,0,0,0,0,0,0,0,0,0,0]),

			(n := [0,0,0,0,0,0,0,0,0,0,0,0,0,0,0,0,0,0,0,0,0,0,0,0,0,0,0,0,0,0,0,0,0,0,0,0,0,0,0,0,0,0,0,0,0,0,0,0,0,0,0,0,0,0,0,0,0,0,0,0,0,0,0,0,0,0,0,0,0,0,0]),
			(n := [0,0,0,0,0,0,0,0,0,0,0,0,0,0,0,0,0,0,0,0,0,0,0,0,0,0,0,0,0,0,0,0,0,0,0,0,0,0,0,0,0,0,0,0,0,0,0,0,0,0,0,0,0,0,0,0,0,0,0,0,0,0,0,0,0,0,0,0,0,0,0]),
			(n := [0,0,0,0,0,0,0,0,0,0,0,0,0,0,0,0,0,0,0,0,0,0,0,0,0,0,0,0,0,0,0,0,0,0,0,0,0,0,0,0,0,0,0,0,0,0,0,0,0,0,0,0,0,0,0,0,0,0,0,0,0,0,0,0,0,0,0,0,0,0,0]),	// SVE
			(n := [0,0,0,0,0,0,0,0,0,0,0,0,0,0,0,0,0,0,0,0,0,0,0,0,0,0,0,0,0,0,0,0,0,0,0,0,0,0,0,0,0,0,0,0,0,0,0,0,0,0,0,0,0,0,0,0,0,0,0,0,0,0,0,0,0,0,0,0,0,0,0]),
			(n := [0,0,0,0,0,0,0,0,0,0,0,0,0,0,0,0,0,0,0,0,0,0,0,0,0,0,0,0,0,0,0,0,0,0,0,0,0,0,0,0,0,0,0,0,0,0,0,0,0,0,0,0,0,0,0,0,0,0,0,0,0,0,0,0,0,0,0,0,0,0,0]),
			(n := [0,0,0,0,0,0,0,0,0,0,0,0,0,0,0,0,0,0,0,0,0,0,0,0,0,0,0,0,0,0,0,0,0,0,0,0,0,0,0,0,0,0,0,0,0,0,0,0,0,0,0,0,0,0,0,0,0,0,0,0,0,0,0,0,0,0,0,0,0,0,0]),	// SVE

			()
			];

   END_STRUCT

   NH_FRM_236     {HIDDEN}    : STRUCT
//      typ : USINT := 236;
      hed : NH_FRM_HED :=(Name:='_236',desc:='Dev-list:ACT,SCN,',wht:=0) ;
		rgbwa	: FILT_LIST := // zoznam DEV (v riadku) ktore maju DLs {vhlavicke) vo svojom HW vratane RGBWA
//                 0         5         10        15        20        25        30        35	      40        45	     50        55	       60        65
				(n := [0,0,0,0,0,0,0,1,1,1,1,1,1,0,0,0,0,0,0,0,0,1,0,1,0,0,0,0,0,0,0,0,1,0,0,0,0,1,0,0,0,0,0,0,0,0,0,0,0,0,0,0,0,0,0,0,0,0,0,0,0,0,0,0,0,0]);     //  HW vazby DLs k DEV vratane RGBWA
      lst : ARRAY[0.._Nh_CFG] OF FILT_LIST := [ // v riadku je DEV z hlavicky a stlpce su DEV ktore mozu byt v LISTE (ACT,SCN,BLK..)
            (),     //  0 prazdne               napr (ACT->GAT,SVx,SCN...)
            (n := [0,0,0,0,0,0,0,0,0,0,0,0,0,0,0,0,0,0,0,0,0,0,0,0,0,0,0,0,0,0,0,0,0,0,0,0,0,0,0,0,0,0,0,0,0,0,0,0,0,0,0,0,0,0,0,0,0,0,0,0,0,0,0,0,0,0]),     //  1 rom  miestnosti (vsetko)
            (n := [0,0,1]),    //  2 cat ... len cat
            (n := [0,1,0]),    //  3 zone/subj - len miestnosti
            // 4                                                                                                                                              //  toto je v HLAVICKE
//                 0         5         10        15        20        25        30        35	      40        45	     50        55	       60        65
            (n := [0,0,0,0,0,0,0,0,0,0,1,1,1,0,0,0,0,0,0,0,0,1,0,0,0,0,0,0,0,0,1,1,1,0,0,1,0,1,0,0,0,0,1,1,1,0,0,0,0,1,0,0,0,0,0,0,0,0,0,0,0,0,0,0,0,0]) ,    //  4 scn  sceny
            (n := [0,0,0,0,1,0,1,0,0,0,1,1,1,0,0,0,0,0,0,0,0,1,0,0,0,0,0,0,0,0,1,1,1,0,0,1,0,1,0,0,0,0,1,1,1,0,0,1,0,1,0,0,0,0,0,0,0,0,0,0,0,0,0,0,0,0]) ,    //  5 act  akcie
            (n := [0,0,0,0,0,1,0,0,0,0,0,0,0,0,0,0,0,0,0,0,0,0,0,0,0,0,0,0,0,0,0,0,0,0,0,0,0,0,0,0,0,0,0,0,0,0,0,0,0,0,0,0,0,0,0,0,0,0,0,0,0,0,0,0,0,0]) ,    //  6 het  modul kurenia
            (n := [0,0,0,0,0,0,0,0,0,0,0,0,0,0,0,0,0,0,0,0,0,0,0,0,0,0,0,0,0,0,0,0,0,0,0,0,0,0,0,0,0,0,0,0,0,0,0,0,0,0,0,0,0,0,0,0,0,0,0,0,0,0,0,0,0,0]) ,    //  7 kot  kotol

            (n := [0,0,0,0,0,0,0,0,0,0,0,0,0,0,0,0,0,0,0,0,0,0,0,0,0,0,0,0,0,0,0,0,0,0,0,0,0,0,0,0,0,0,0,0,0,0,0,0,0,0,0,0,0,0,0,0,0,0,0,0,0,0,0,0,0,0]) ,    //  8 TVE  termoventil,spirala
            (n := [0,0,0,0,0,0,0,0,0,0,0,0,0,0,0,0,0,0,0,0,0,0,0,0,0,0,0,0,0,0,0,0,0,0,0,0,0,0,0,0,0,0,0,0,0,0,0,0,0,0,0,0,0,0,0,0,0,0,0,0,0,0,0,0,0,0]) ,    //  9 CER  obehove cerpadlo
            (n := [0,0,0,0,1,1,0,0,0,0,0,0,0,0,0,0,0,0,0,0,0,0,0,0,0,0,0,0,0,0,0,0,0,0,0,1,0,0,0,0,0,0,0,0,0,0,0,0,0,0,0,0,0,0,0,0,0,0,0,0,0,0,0,0,0,0]) ,    // 10 SVD  svetlo digital
            (n := [0,0,0,0,1,1,0,0,0,0,0,0,0,0,0,0,0,0,0,0,0,0,0,0,0,0,0,0,0,0,0,0,0,0,0,1,0,0,0,0,0,0,0,0,0,0,0,0,0,0,0,0,0,0,0,0,0,0,0,0,0,0,0,0,0,0]) ,    // 11 SVA  svetlo stivatelne
            (n := [0,0,0,0,1,1,0,0,0,0,0,0,0,0,0,0,0,0,0,0,0,0,0,0,0,0,0,0,0,0,0,0,0,0,0,1,0,0,0,0,0,0,0,0,0,0,0,0,0,0,0,0,0,0,0,0,0,0,0,0,0,0,0,0,0,0]) ,    // 12 RGB  svetlo farebne
            (n := [0,0,0,0,0,1,1,0,0,0,1,1,1,0,0,0,0,0,0,0,0,1,0,1,0,0,0,0,0,0,1,1,0,0,0,1,0,1,0,0,0,0,1,1,0,0,0,0,0,0,0,0,0,0,0,0,0,0,0,1,0,0,0,0,0,0]) ,    // 13 WSB  ovladac WSB
            (n := [0,0,0,0,0,1,0,0,0,0,1,1,1,0,0,0,0,0,0,0,0,1,0,1,0,0,0,0,0,0,1,1,0,0,0,1,0,1,0,0,0,0,1,1,0,0,0,0,0,0,0,0,0,0,0,0,0,0,0,1,0,0,0,0,0,0]) ,    // 14 TLA  tlacitka
            (n := [0,0,0,0,0,1,0,0,0,0,1,1,1,0,0,0,0,0,0,0,0,1,0,1,0,0,0,0,0,0,0,0,1,0,0,1,0,0,0,0,0,0,0,1,1,0,0,0,0,1,0,0,0,0,0,0,0,0,0,0,0,0,0,0,0,0]) ,    // 15 pir
            (n := [0,0,0,0,0,0,1,0,0,0,0,0,0,0,0,0,0,0,0,0,0,0,0,0,0,0,0,0,0,0,0,0,0,0,0,0,0,0,0,0,0,0,0,0,0,0,0,0,0,1,0,0,0,0,0,0,0,0,0,0,0,0,0,0,0,0]) ,    // 16 teR  teplota-miestnost
            (n := [0,0,0,0,0,0,0,0,0,0,0,0,0,0,0,0,0,0,0,0,0,0,0,0,0,0,0,0,0,0,0,0,0,0,0,0,0,0,0,0,0,0,0,0,0,0,0,0,0,1,0,0,0,0,0,0,0,0,0,0,0,0,0,0,0,0]) ,    // 17 teH  teplota-teleso
            (n := [0,0,0,0,0,0,0,0,0,0,0,0,0,0,0,0,0,0,0,0,0,0,0,0,0,0,0,0,0,0,0,0,0,0,0,0,0,0,0,0,0,0,0,0,0,0,0,0,0,0,0,0,0,0,0,0,0,0,0,0,0,0,0,0,0,0]) ,    // 18 teK  teplota-kotol
            (n := [0,0,0,0,0,0,0,0,0,0,0,0,0,0,0,0,0,0,0,0,0,0,0,0,0,0,0,0,0,0,0,0,0,0,0,0,0,0,0,0,0,0,0,0,0,0,0,0,0,0,0,0,0,0,0,0,0,0,0,0,0,0,0,0,0,0]) ,    // 19 lux  intenzita osvetlenia
            (n := [0,0,0,0,0,0,0,0,0,0,0,0,0,0,0,0,0,0,0,0,0,0,0,0,0,0,0,0,0,0,0,0,0,0,0,0,0,0,0,0,0,0,0,0,0,0,0,0,0,1,0,0,0,0,0,0,0,0,0,0,0,0,0,0,0,0]) ,    // 20 FAV
            (n := [0,0,0,0,1,1,0,0,0,0,0,0,0,0,0,0,0,0,0,0,0,0,0,0,0,0,0,0,0,0,0,0,0,0,0,1,0,0,0,0,0,0,0,0,0,0,0,0,0,0,0,0,0,0,0,0,0,0,0,0,0,0,0,0,0,0]) ,    // 21 ZAS  spotrebice
            (n := [0,0,0,0,0,0,0,0,0,0,0,0,0,0,0,0,0,0,0,0,0,0,0,0,0,0,0,0,0,0,0,0,0,0,0,0,0,0,0,0,0,0,0,0,0,0,0,0,0,1,0,0,0,0,0,0,0,0,0,0,0,0,0,0,0,0]) ,    // 22 USR  uzivatelia
            (n := [0,0,0,0,0,0,0,0,0,0,0,0,0,0,0,0,0,0,0,0,0,0,0,0,0,0,0,0,0,0,0,0,0,0,0,0,0,0,0,0,0,0,0,0,0,0,0,1,0,0,0,0,0,0,0,0,0,0,0,0,0,0,0,0,0,0]) ,    // 23 VENT+REK-uperacia
            (n := [0,0,0,0,0,0,0,0,0,0,0,0,0,0,0,0,0,0,0,0,0,0,0,0,0,0,0,0,0,0,0,0,0,0,0,0,0,0,0,0,0,0,0,0,0,0,0,0,0,1,0,0,0,0,0,0,0,0,0,0,0,0,0,0,0,0]),     // 24 KEY
            (n := [0,0,0,0,0,0,0,0,0,0,0,0,0,0,0,0,0,0,0,0,0,0,0,0,0,0,0,0,0,0,0,0,0,0,0,0,0,0,0,0,0,0,0,0,0,0,0,0,0,1,0,0,0,0,0,0,0,0,0,0,0,0,0,0,0,0]),     // 25 RZV - casovy rozvrh PO-NE
            (n := [0,0,0,0,0,0,0,0,0,0,0,0,0,0,0,0,0,0,0,0,0,0,0,0,0,0,0,0,0,0,0,0,0,0,0,0,0,0,0,0,0,0,0,0,0,0,0,0,0,1,0,0,0,0,0,0,0,0,0,0,0,0,0,0,0,0]),     // 26 POI - slider
            (n := [0,0,0,0,0,0,0,0,0,0,0,0,0,0,0,0,0,0,0,0,0,0,0,0,0,0,0,0,0,0,0,0,0,0,0,0,0,0,0,0,0,0,0,0,0,0,0,0,0,1,0,0,0,0,0,0,0,0,0,0,0,0,0,0,0,0]),     // 27 H2O
            (n := [0,0,0,0,0,0,0,0,0,0,0,0,0,0,0,0,0,0,0,0,0,0,0,0,0,0,0,0,0,0,0,0,0,0,0,0,0,0,0,0,0,0,0,0,0,0,0,0,0,1,0,0,0,0,0,0,0,0,0,0,0,0,0,0,0,0]),     // 28 FIRe - len ON/OFF : poziar,dym,CO,CO2,butan...
            (n := [0,0,0,0,0,0,0,0,0,0,0,0,0,0,0,0,0,0,0,0,0,0,0,0,0,0,0,0,0,0,0,0,0,0,0,0,0,0,0,0,0,0,0,0,0,0,0,0,0,1,0,0,0,0,0,0,0,0,0,0,0,0,0,0,0,0]),     // 29 GAS // intenzita (real) CO,CO2,metan,butan,RH
            (n := [0,0,0,0,0,1,0,0,0,0,0,0,0,1,1,0,0,0,0,0,0,0,0,0,0,0,0,0,0,0,0,0,0,0,0,0,0,0,0,0,1,0,0,0,0,0,0,0,0,0,0,0,0,0,0,0,0,0,0,1,0,0,0,0,0,0]),     // 30 MAR garaz,brana,branicka
            (n := [0,0,0,0,0,1,0,0,0,0,0,0,0,1,1,0,0,0,0,0,0,0,0,0,0,0,0,0,0,0,0,0,0,0,0,0,0,0,0,0,1,0,0,0,0,0,0,0,0,0,0,0,0,0,0,0,0,0,0,1,0,0,0,0,0,0]),     // 31 ROL rolety
            (n := [0,0,0,0,1,1,0,0,0,0,0,0,0,1,1,1,0,0,0,0,0,0,0,0,0,0,0,0,0,0,0,0,0,0,0,1,0,0,0,0,1,0,0,0,0,0,0,0,0,0,0,0,0,0,0,0,0,0,0,1,0,0,0,0,0,0]),     // 32 SIR sirena,stroboskop,zvoncek
            (n := [0,0,0,0,0,0,0,0,0,0,0,0,0,0,0,0,0,0,0,0,0,0,0,0,0,0,0,0,0,0,0,0,0,0,0,0,0,1,0,0,0,0,0,0,0,0,0,0,0,0,0,0,0,0,0,0,0,0,0,0,0,0,0,0,0,0]),     // 33 DOR
            (n := [0,0,0,0,0,0,0,0,0,0,0,0,0,0,0,0,0,0,0,0,0,0,0,0,0,0,0,0,0,0,0,0,0,0,0,0,0,1,0,0,0,0,0,0,0,0,0,0,0,0,0,0,0,0,0,0,0,0,0,0,0,0,0,0,0,0]),     // 34 WIN
//                 0         5         10        15        20        25        30        35	      40        45	     50        55	       60        65
            (n := [0,0,0,0,1,0,0,0,0,0,1,1,1,0,0,0,0,0,0,0,0,1,0,0,0,0,0,0,0,0,0,0,1,0,0,0,0,0,0,0,0,0,1,1,1,0,0,0,0,0,0,0,0,0,0,0,0,0,0,0,0,0,0,0,0,0]),     // 35 BLK
            (n := [0,0,0,0,0,0,0,0,0,0,0,0,0,0,0,0,0,0,0,0,0,0,0,0,0,0,0,0,0,0,0,0,0,0,0,0,0,0,0,0,0,0,0,0,0,0,0,0,0,1,0,0,0,0,0,0,0,0,0,0,0,0,0,0,0,0]),     // 36    XXX*BLx
            (n := [0,0,0,0,0,0,0,0,0,0,0,0,0,0,0,0,0,0,0,0,0,0,0,0,0,0,0,0,0,0,0,0,0,1,1,0,0,0,0,0,0,0,0,0,0,0,0,0,0,0,0,0,0,0,0,0,0,0,0,0,0,0,0,0,0,0]),     // 37 BRA,GAR....
            (n := [0,0,0,0,1,1,0,0,0,0,0,0,0,0,0,0,0,0,0,0,0,0,0,0,0,0,0,0,0,0,0,0,0,0,0,0,0,0,0,0,0,0,0,0,0,0,0,0,0,1,0,0,0,0,0,0,0,0,0,0,0,0,0,0,0,0]),     // 38 RFI
            (n := [0,0,0,0,1,1,0,0,0,0,0,0,0,0,0,0,0,0,0,0,0,0,0,0,0,0,0,0,0,0,0,0,0,0,0,0,0,0,0,0,0,0,0,0,0,0,0,0,0,1,0,0,0,0,0,0,0,0,0,0,0,0,0,0,0,0]),     // 39 RFK
            (n := [0,0,0,0,1,1,1,0,0,0,1,1,1,0,0,0,0,0,0,0,0,0,0,1,0,0,0,0,0,0,1,1,0,0,0,1,0,1,0,0,0,0,1,1,0,0,0,0,0,0,0,0,0,0,0,0,0,0,0,1,0,0,0,0,0,0]),     // 40 TGL
            (n := [0,0,0,0,1,1,0,0,0,0,0,0,0,0,0,0,0,0,0,0,0,0,0,0,0,0,0,0,0,0,0,0,0,0,0,0,0,0,0,0,0,0,0,0,0,0,0,0,0,1,0,0,0,0,0,0,0,0,0,0,0,0,0,0,0,0]),     // 41 COX
            (n := [0,0,0,0,1,1,0,0,0,0,0,0,0,0,0,0,0,0,0,0,0,0,0,0,0,0,0,0,0,0,0,0,0,0,0,0,0,0,0,0,0,0,0,0,0,0,0,0,0,1,0,0,0,0,0,0,0,0,0,0,0,0,0,0,0,0]),     // 42 DALI*M
            (n := [0,0,0,0,1,1,0,0,0,0,0,0,0,0,0,0,0,0,0,0,0,0,0,0,0,0,0,0,0,0,0,0,0,0,0,0,0,0,0,0,0,0,0,0,1,0,0,0,0,0,0,0,0,0,0,0,0,0,0,0,0,0,0,0,0,0]),     // 43 DALI - S
            (n := [0,0,0,0,0,0,0,0,0,0,0,0,0,0,0,0,0,0,0,0,0,0,0,0,0,0,0,0,0,0,0,0,0,0,0,0,0,0,0,0,0,0,0,1,0,0,0,0,0,0,0,0,0,0,0,0,0,0,0,0,0,0,0,0,0,0]),     // 44 DALI - GRP
            (n := [0,0,0,0,0,0,0,0,0,0,0,0,0,0,0,0,0,0,0,0,0,0,0,0,0,0,0,0,0,0,0,0,0,0,0,0,0,0,0,0,0,0,0,0,0,0,0,0,0,1,0,0,0,0,0,0,0,0,0,0,0,0,0,0,0,0]),     // 45 SMW - smart way
//                 0         5         10        15        20        25        30        35	      40        45	     50        55	       60        65
            (n := [0,0,0,0,0,0,0,0,0,0,0,0,0,0,0,0,0,0,0,0,0,0,0,0,0,0,0,0,0,0,0,0,0,0,0,0,0,0,0,0,0,0,0,0,0,0,0,0,0,0,0,0,0,0,0,0,0,0,0,0,0,0,0,0,0,0]),     // 46 MSG
            (n := [0,0,0,0,0,1,0,0,0,0,0,0,0,0,0,0,0,0,0,0,0,0,0,0,0,0,0,0,0,0,0,0,0,0,0,0,0,0,0,0,0,0,0,0,0,0,0,0,0,0,0,0,0,0,0,0,0,0,0,0,0,0,0,0,0,0]),     // 47 HEV {HET pre vetranie}
            (n := [0,0,0,0,1,1,0,0,0,0,0,0,0,0,0,0,0,0,0,0,0,0,0,0,0,0,0,0,0,0,0,0,1,0,0,1,0,0,0,0,0,0,0,0,0,0,0,0,0,1,0,0,0,0,0,0,0,0,0,0,0,0,0,0,0,0]),     // 48 ALA akce ALArmu
            (n := [0,0,0,0,0,0,0,0,0,0,0,0,0,0,0,0,0,0,0,0,0,0,0,0,0,0,0,0,0,0,0,0,0,0,0,0,0,0,0,0,0,0,0,0,0,0,0,0,0,0,0,0,0,0,0,0,0,0,0,0,0,0,0,0,0,0])      // 49 VVO
         ];
				  // vazby dev , externe vazby, HET,HEV ....
      iodev : ARRAY[0.._Nh_CFG] OF FILT_LIST := [ // v riadku je DEV z hlavicky a stlpce su DEV ktore mozu byt v LISTE (ACT,SCN,BLK..)
            (),     //  0 prazdne               napr (ACT->GAT,SVx,SCN...)
            (n := [0,0,0,0,0,0,0,0,0,0,0,0,0,0,0,0,0,0,0,0,0,0,0,0,0,0,0,0,0,0,0,0,0,0,0,0,0,0,0,0,0,0,0,0,0,0,0,0,0,0,0,0,0,0,0,0,0,0,0,0,0,0,0,0,0,0]),        //  1 rom  miestnosti (vsetko)
            (n := [0,0,1]),    //  2 cat ... len cat
            (n := [0,1,0]),    //  3 zone/subj - len miestnosti
            // 4                                                                                                                                              //  toto je v HLAVICKE
//                 0         5         10        15        20        25        30        35	      40        45	     50        55	       60        65
            (n := [0,0,0,0,0,0,0,0,0,0,1,1,1,0,0,0,0,0,0,0,0,1,0,0,0,0,0,0,0,0,1,1,1,0,0,1,0,1,0,0,0,0,1,1,1,0,0,0,0,0,0,0,0,0,0,0,0,0,0,0,0,0,0,0,0,0]) ,    //  4 scn  sceny
            (n := [0,0,0,0,1,0,1,0,0,0,1,1,1,0,0,0,0,0,0,0,0,1,0,0,0,0,0,0,0,0,1,1,1,0,0,1,0,1,0,0,0,0,1,1,1,0,0,0,0,0,0,0,0,0,0,0,0,0,0,0,0,0,0,0,0,0]) ,    //  5 act  akcie
            (n := [0,1,0,0,0,0,0,1,1,1,0,0,0,0,0,0,1,1,1,0,0,0,0,0,0,0,0,0,0,0,0,0,0,0,0,0,0,0,0,0,0,0,0,0,0,0,0,0,0,0,0,0,0,0,0,0,0,0,0,0,0,0,0,0,0,0]) ,    //  6 het  modul kurenia
            (n := [0,0,0,0,0,0,0,0,0,0,0,0,0,0,0,0,0,0,1,0,0,0,0,0,0,0,0,0,0,0,0,0,0,0,0,0,0,0,0,0,0,0,0,0,0,0,0,0,0,0,0,0,0,0,0,0,0,0,0,0,0,0,0,0,0,0]) ,    //  7 kot  kotol

            (n := [0,0,0,0,0,0,0,0,0,0,0,0,0,0,0,0,0,1,0,0,0,0,0,0,0,0,0,0,0,0,0,0,0,0,0,0,0,0,0,0,0,0,0,1,0,0,0,0,0,0,0,0,0,0,0,0,0,0,0,0,0,0,0,0,0,0]) ,    //  8 TVE  termoventil,spirala
            (n := [0,0,0,0,0,0,0,0,0,0,0,0,0,0,0,0,0,0,1,0,0,0,0,0,0,0,0,0,0,0,0,0,0,0,0,0,0,0,0,0,0,0,0,0,0,0,0,0,0,0,0,0,0,0,0,0,0,0,0,0,0,0,0,0,0,0]) ,    //  9 CER  obehove cerpadlo
            (n := [0,0,0,0,1,1,0,0,0,0,0,0,0,0,0,0,0,0,0,0,0,0,0,0,0,0,0,0,0,0,0,0,0,0,0,1,0,0,0,0,0,0,0,0,0,0,0,0,0,0,0,0,0,0,0,0,0,0,0,0,0,0,0,0,0,0]) ,    // 10 SVD  svetlo digital
            (n := [0,0,0,0,1,1,0,0,0,0,0,0,0,0,0,0,0,0,0,0,0,0,0,0,0,0,0,0,0,0,0,0,0,0,0,1,0,0,0,0,0,0,0,0,0,0,0,0,0,0,0,0,0,0,0,0,0,0,0,0,0,0,0,0,0,0]) ,    // 11 SVA  svetlo stivatelne
            (n := [0,0,0,0,1,1,0,0,0,0,0,0,0,0,0,0,0,0,0,0,0,0,0,0,0,0,0,0,0,0,0,0,0,0,0,1,0,0,0,0,0,0,0,0,0,0,0,0,0,0,0,0,0,0,0,0,0,0,0,0,0,0,0,0,0,0]) ,    // 12 RGB  svetlo farebne
            (n := [0,0,0,0,1,1,1,0,0,0,1,1,1,0,0,0,0,0,0,0,0,1,0,1,0,0,0,0,0,0,1,1,0,0,0,1,0,1,0,0,0,0,1,1,0,0,0,0,0,0,0,0,0,0,0,0,0,0,0,1,0,0,0,0,0,0]) ,    // 13 WSB  ovladac WSB
            (n := [0,0,0,0,1,1,0,0,0,0,1,1,1,0,0,0,0,0,0,0,0,1,0,1,0,0,0,0,0,0,1,1,0,0,0,1,0,1,0,0,0,0,1,1,0,0,0,0,0,0,0,0,0,0,0,0,0,0,0,1,0,0,0,0,0,0]) ,    // 14 TLA  tlacitka
            (n := [0,0,0,0,1,1,0,0,0,0,1,1,1,0,0,0,0,0,0,0,0,1,0,1,0,0,0,0,0,0,0,0,1,0,0,1,0,0,0,0,0,0,0,1,1,0,0,0,0,1,0,0,0,0,0,0,0,0,0,0,0,0,0,0,0,0]) ,    // 15 pir
            (n := [0,0,0,1,0,0,1,0,0,0,0,0,0,0,0,0,0,0,0,0,0,0,0,0,0,0,0,0,0,0,0,0,0,0,0,0,0,0,0,0,0,0,0,0,0,0,0,0,0,1,0,0,0,0,0,0,0,0,0,0,0,0,0,0,0,0]) ,    // 16 teR  teplota-miestnost
            (n := [0,0,0,0,0,0,1,0,1,0,0,0,0,0,0,0,0,0,0,0,0,0,0,0,0,0,0,0,0,0,0,0,0,0,0,0,0,0,0,0,0,0,0,0,0,0,0,0,0,1,0,0,0,0,0,0,0,0,0,0,0,0,0,0,0,0]) ,    // 17 teH  teplota-teleso
            (n := [0,0,0,0,0,0,1,1,0,0,0,0,0,0,0,0,0,0,0,0,0,0,0,0,0,0,0,0,0,0,0,0,0,0,0,0,0,0,0,0,0,0,0,0,0,0,0,0,0,0,0,0,0,0,0,0,0,0,0,0,0,0,0,0,0,0]) ,    // 18 teK  teplota-kotol
            (n := [0,0,0,1,0,0,0,0,0,0,0,0,0,0,0,0,0,0,0,0,0,0,0,0,0,0,0,0,0,0,0,0,0,0,0,0,0,0,0,0,0,0,0,0,0,0,0,0,0,0,0,0,0,0,0,0,0,0,0,0,0,0,0,0,0,0]) ,    // 19 lux  intenzita osvetlenia
            (n := [0,0,0,0,0,0,0,0,0,0,0,0,0,0,0,0,0,0,0,0,0,0,0,0,0,0,0,0,0,0,0,0,0,0,0,0,0,0,0,0,0,0,0,0,0,0,0,0,0,1,0,0,0,0,0,0,0,0,0,0,0,0,0,0,0,0]) ,    // 20 FAV
            (n := [0,0,0,0,1,1,0,0,0,0,0,0,0,0,0,0,0,0,0,0,0,0,0,0,0,0,0,0,0,0,0,0,0,0,0,1,0,0,0,0,0,0,0,0,0,0,0,0,0,0,0,0,0,0,0,0,0,0,0,0,0,0,0,0,0,0]) ,    // 21 ZAS  spotrebice
            (n := [0,0,0,0,0,0,0,0,0,0,0,0,0,0,0,0,0,0,0,0,0,0,0,0,0,0,0,0,0,0,0,0,0,0,0,0,0,0,0,0,0,0,0,0,0,0,0,0,0,1,0,0,0,0,0,0,0,0,0,0,0,0,0,0,0,0]) ,    // 22 USR  uzivatelia
            (n := [0,0,0,0,0,0,0,0,0,0,0,0,0,0,0,0,0,0,0,0,0,0,0,0,0,0,0,0,0,0,0,0,0,0,0,0,0,0,0,0,0,0,0,1,0,0,0,0,0,0,0,0,0,0,0,0,0,0,0,0,0,0,0,0,0,0]) ,    // 23 VEN+REK-uperacia
            (n := [0,0,0,0,0,0,0,0,0,0,0,0,0,0,0,0,0,0,0,0,0,0,0,0,0,0,0,0,0,0,0,0,0,0,0,0,0,0,0,0,0,0,0,0,0,0,0,0,0,1,0,0,0,0,0,0,0,0,0,0,0,0,0,0,0,0]),     // 24 KEY
            (n := [0,0,0,0,0,0,0,0,0,0,0,0,0,0,0,0,0,0,0,0,0,0,0,0,0,0,0,0,0,0,0,0,0,0,0,0,0,0,0,0,0,0,0,0,0,0,0,0,0,1,0,0,0,0,0,0,0,0,0,0,0,0,0,0,0,0]),     // 25 RZV - casovy rozvrh PO-NE
            (n := [0,0,0,0,0,0,0,0,0,0,0,0,0,0,0,0,0,0,0,0,0,0,0,0,0,0,0,0,0,0,0,0,0,0,0,0,0,0,0,0,0,0,0,0,0,0,0,0,0,1,0,0,0,0,0,0,0,0,0,0,0,0,0,0,0,0]),     // 26 POI - slider
            (n := [0,0,0,0,0,0,0,0,0,0,0,0,0,0,0,0,0,0,0,0,0,0,0,0,0,0,0,0,0,0,0,0,0,0,0,0,0,0,0,0,0,0,0,0,0,0,0,0,0,1,0,0,0,0,0,0,0,0,0,0,0,0,0,0,0,0]),     // 27 H2O
            (n := [0,0,0,0,0,0,0,0,0,0,0,0,0,0,0,0,0,0,0,0,0,0,0,0,0,0,0,0,0,0,0,0,0,0,0,0,0,0,0,0,0,0,0,0,0,0,0,0,0,1,0,0,0,0,0,0,0,0,0,0,0,0,0,0,0,0]),     // 28 FIRe - len ON/OFF : poziar,dym,CO,CO2,butan...
            (n := [0,0,0,0,0,0,0,0,0,0,0,0,0,0,0,0,0,0,0,0,0,0,0,0,0,0,0,0,0,0,0,0,0,0,0,0,0,0,0,0,0,0,0,0,0,0,0,0,0,1,0,0,0,0,0,0,0,0,0,0,0,0,0,0,0,0]),     // 29 GAS // intenzita (real) CO,CO2,metan,butan,RH
            (n := [0,0,0,0,0,0,0,0,0,0,0,0,0,1,1,0,0,0,0,0,0,0,0,0,0,0,0,0,0,0,0,0,0,0,0,0,0,0,0,0,1,0,0,0,0,0,0,0,0,0,0,0,0,0,0,0,0,0,0,1,0,0,0,0,0,0]),     // 30 MAR garaz,brana,branicka
            (n := [0,0,0,0,0,0,0,0,0,0,0,0,0,1,1,0,0,0,0,0,0,0,0,0,0,0,0,0,0,0,0,0,0,0,0,0,0,0,0,0,1,0,0,0,0,0,0,0,0,0,0,0,0,0,0,0,0,0,0,1,0,0,0,0,0,0]),     // 31 ROL rolety
            (n := [0,0,0,0,0,0,0,0,0,0,0,0,0,1,1,1,0,0,0,0,0,0,0,0,0,0,0,0,0,0,0,0,0,0,0,1,0,0,0,0,1,0,0,0,0,0,0,0,0,0,0,0,0,0,0,0,0,0,0,1,0,0,0,0,0,0]),     // 32 SIR sirena,stroboskop,zvoncek
            (n := [0,0,0,0,0,0,0,0,0,0,0,0,0,0,0,0,0,0,0,0,0,0,0,0,0,0,0,0,0,0,0,0,0,0,0,0,0,1,0,0,0,0,0,0,0,0,0,0,0,0,0,0,0,0,0,0,0,0,0,0,0,0,0,0,0,0]),     // 33 DOR
            (n := [0,0,0,0,0,0,0,0,0,0,0,0,0,0,0,0,0,0,0,0,0,0,0,0,0,0,0,0,0,0,0,0,0,0,0,0,0,1,0,0,0,0,0,0,0,0,0,0,0,0,0,0,0,0,0,0,0,0,0,0,0,0,0,0,0,0]),     // 34 WIN
//                 0         5         10        15        20        25        30        35	      40        45	     50        55	       60        65
            (n := [0,0,0,0,1,1,0,0,0,0,1,1,1,0,0,0,0,0,0,0,0,1,0,0,0,0,0,0,0,0,0,0,1,0,0,0,0,0,0,0,0,0,1,1,1,0,0,0,0,0,0,0,0,0,0,0,0,0,0,0,0,0,0,0,0,0]),     // 35 BLK
            (n := [0,0,0,0,0,0,0,0,0,0,0,0,0,0,0,0,0,0,0,0,0,0,0,0,0,0,0,0,0,0,0,0,0,0,0,0,0,0,0,0,0,0,0,0,0,0,0,0,0,1,0,0,0,0,0,0,0,0,0,0,0,0,0,0,0,0]),     // 36    XXX*BLx
            (n := [0,0,0,0,0,0,0,0,0,0,0,0,0,0,0,0,0,0,0,0,0,0,0,0,0,0,0,0,0,0,0,0,0,1,1,0,0,0,0,0,0,0,0,0,0,0,0,0,0,0,0,0,0,0,0,0,0,0,0,0,0,0,0,0,0,0]),     // 37 BRA,GAR....
            (n := [0,0,0,0,1,1,0,0,0,0,0,0,0,0,0,0,0,0,0,0,0,0,0,0,0,0,0,0,0,0,0,0,0,0,0,0,0,0,0,0,0,0,0,0,0,0,0,0,0,1,0,0,0,0,0,0,0,0,0,0,0,0,0,0,0,0]),     // 38 RFI
            (n := [0,0,0,0,1,1,0,0,0,0,0,0,0,0,0,0,0,0,0,0,0,0,0,0,0,0,0,0,0,0,0,0,0,0,0,0,0,0,0,0,0,0,0,0,0,0,0,0,0,1,0,0,0,0,0,0,0,0,0,0,0,0,0,0,0,0]),     // 39 RFK
            (n := [0,0,0,0,1,1,1,0,0,0,1,1,1,0,0,0,0,0,0,0,0,0,0,1,0,0,0,0,0,0,1,1,0,0,0,1,0,1,0,0,0,0,1,1,0,0,0,0,0,0,0,0,0,0,0,0,0,0,0,1,0,0,0,0,0,0]),     // 40 TGL
            (n := [0,0,0,0,1,1,0,0,0,0,0,0,0,0,0,0,0,0,0,0,0,0,0,0,0,0,0,0,0,0,0,0,0,0,0,0,0,0,0,0,0,0,0,0,0,0,0,0,0,1,0,0,0,0,0,0,0,0,0,0,0,0,0,0,0,0]),     // 41 COX
            (n := [0,0,0,0,1,1,0,0,0,0,0,0,0,0,0,0,0,0,0,0,0,0,0,0,0,0,0,0,0,0,0,0,0,0,0,0,0,0,0,0,0,0,0,0,0,0,0,0,0,1,0,0,0,0,0,0,0,0,0,0,0,0,0,0,0,0]),     // 42 DALI*M
            (n := [0,0,0,0,0,0,0,0,0,0,0,0,0,0,0,0,0,0,0,0,0,0,0,0,0,0,0,0,0,0,0,0,0,0,0,0,0,0,0,0,0,0,0,0,1,0,0,0,0,0,0,0,0,0,0,0,0,0,0,0,0,0,0,0,0,0]),     // 43 DALI - S
            (n := [0,0,0,0,0,0,0,0,0,0,0,0,0,0,0,0,0,0,0,0,0,0,0,0,0,0,0,0,0,0,0,0,0,0,0,0,0,0,0,0,0,0,0,1,0,0,0,0,0,0,0,0,0,0,0,0,0,0,0,0,0,0,0,0,0,0]),     // 44 DALI - GRP
            (n := [0,0,0,0,1,1,0,0,0,0,0,0,0,0,0,0,0,0,0,0,0,0,0,0,0,0,0,0,0,0,0,0,0,0,0,0,0,0,0,0,0,0,0,0,0,0,0,0,0,1,0,0,0,0,0,0,0,0,0,0,0,0,0,0,0,0]),     // 45 SMW - smart way
//                 0         5         10        15        20        25        30        35	      40        45	     50        55	       60        65
            (n := [0,0,0,0,0,0,0,0,0,0,0,0,0,0,0,0,0,0,0,0,0,0,0,0,0,0,0,0,0,0,0,0,0,0,0,0,0,0,0,0,0,0,0,0,0,0,0,0,0,0,0,0,0,0,0,0,0,0,0,0,0,0,0,0,0,0]),     // 46 MSG
            (n := [0,0,0,0,0,0,0,0,0,0,0,0,0,0,0,0,0,0,0,0,0,0,0,1,0,0,0,0,0,0,0,0,0,0,0,0,0,0,0,0,0,1,0,0,0,0,0,0,0,0,0,0,0,0,0,0,0,0,0,0,0,0,0,0,0,0]),      // 47 HEV {HET pre vetranie}
            (n := [0,0,0,0,0,0,0,0,0,0,0,0,0,0,0,0,0,0,0,0,0,0,0,0,0,0,0,0,0,0,0,0,1,0,0,1,0,0,0,0,0,0,0,0,0,0,0,0,0,0,0,0,0,0,0,0,0,0,0,0,0,0,0,0,0,0])      // 48 HEV akce ALArmu
         ];
   END_STRUCT

   NH_RUN_VAL2_D  {HIDDEN} :  STRUCT          // STAVOVY dash S OBRAZKOM/TEXTOM/HODNOTOU
      ok       : BOOL;
      xy       : BOOL;                    // znamena, ze sa text vypisuje len pre to co je v x,y, inak pre xO^.x + x
      noxy     : BOOL;                    // text sa vypise od nastavenej pozicie
      nofmt    : BOOL;                    // text sa neformatuje
      crc      : BOOL;                    // vykresluje sa kruh
      box      : BOOL;                    // vykresluje sa obdlznik
      fil      : BOOL := true;            // vykresluje sa obsah kruhu/obdlznika
      wh       : USINT;                   // predvolba
      obr      : INT;
      txt      : SINT   := -1;            // vypise sa text (-1 := nic sa nevypise)
      grd      : USINT;                   // typ gradientu
      wO       : INT;
      wC       : INT;
      wB       : INT;                     // vyska boxu
      wT       : INT    := 24;            // velkost textu
      FgC      : USINT  := 2;             // GCOLOR_LTGRAY;
      BgC      : USINT  := 1;             // GCOLOR_BLACK;
      FgT      : USINT  := 4;             // GCOLOR_WHILE;
      fmt      : INT    := 2;             // formatovanie textu (stred riadka, stred textu)
      x,y      : INT;                     // korekcie
      ob       : SINT   := -1;            // > 1 aj namapuje nanovo obj
      val      : STRING[10];
	END_STRUCT;

   NH_RUN_VAL2  {HIDDEN} :  STRUCT          // STAVOVY dash S OBRAZKOM/TEXTOM/HODNOTOU
      v        : ARRAY[0.._ShwVal] OF NH_RUN_VAL2_D := [(ok:=1,wh:=18)];
	END_STRUCT;

	NH_DSH_OBJ	{HIDDEN} :  STRUCT
      rws            : USINT;
      clm            : USINT;
	END_STRUCT;

   NH_DSH	{HIDDEN} :  STRUCT
		dsh 				: ARRAY[0..4] OF NH_DSH_OBJ := [
										( rws := 9,	clm := 1 ),				// home page
										( rws := 7,	clm := 1 ),          // browser - riadok
										( rws := 6,	clm := 2 ),          // brows - velky dash
										( rws :=14,	clm := 2 ),          // brows - maly dash
										( rws :=14,	clm := 1 )];         // brows - tenke riadky pre CHECK
	END_STRUCT;

  	NH_ROW_H  {HIDDEN}  :  STRUCT       // hlavicka RIADKA
      cf       : NH_DEV_IO;                           // cf,nd,par
      nd       : INT;                                 // fyzicke poradove cislo vety v CFG
      sld      : BOOL;                                // ma slider (cislo slider je to iste ako cislo riadka)
      in       : BOOL;                                // tato veta je vo vazbe v xVaz^.in
      btn      : BOOL;                                // priznak, ze nad WSB treba zobrazit BTN, ktory jestlaceny, alebo nakonfigurovany
      chk      : BOOL;                                // zaskrtnuty CHK v riadku - pre Vaz[2]
      dlg      : BOOL;                                // v riadku je vazba DALI sceny -> dalia slave > DLg->DLs
//      del      : BOOL;                                // tento riadok ma objekt del/copy
		pir		: BOOL;											// v riadku je pir
		new      : BOOL;											// uz bola natiahnuta definica, riadi sa teraz druhom refreshu
   END_STRUCT

	NH_POI_DAYWRK {HIDDEN}: NH_POI := ( cx := ( p:= [         // DayMode  Jeden pracovny den
                           ( t :=   0,  o := 2),   // night    0:00
                           ( t := 330,  o := 3),   // morning  5:30 //330
                           ( t := 390,  o := 0),   // day      6:30
                           ( t :=1080,  o := 1),   // evening 18:00
                           ( t :=1380,  o := 2),   // 23:0;
                           ( t :=1440,  o := 2)    // 24:0;
                   ]));
   NH_POI_DAYFRE  {HIDDEN} : NH_POI := ( cx := ( p:= [        // sobota/nedela/sviatok
                           ( t :=   0,  o := 2),   // night    0:00
                           ( t := 450,  o := 3),   // morning  7:30  //450
                           ( t := 480,  o := 0),   // day      8:00
                           ( t :=1080,  o := 1),   // evening 18:00
                           ( t :=1440,  o := 1)    // 24:0;
                   ]));

  	NH_POI_WDAY {HIDDEN}:  STRUCT
      PON       : NH_POI_DAYWRK ;                  // pondelok
      UTO       : NH_POI_DAYWRK ;                  // utorok
      STR       : NH_POI_DAYWRK ;                  // streda
      STV       : NH_POI_DAYWRK ;                  // stvrtok
      PIA       : NH_POI_DAYWRK ;                  // piatok
      SOB       : NH_POI_DAYFRE ;                  // sobota
      NED       : NH_POI_DAYFRE ;                  // nedela
      FRE       : NH_POI_DAYFRE ;                  // volny den /sviatok
      ALL       : NH_POI := ( cx := ( p:= [        // plny dom (party)
                           ( t :=   0,  o := 1),   // night    0:00
                           ( t :=  60,  o := 2),    // 24:0;
                           ( t := 480,  o := 3),   // morning  8:00
                           ( t := 540,  o := 0),   // day      9:00
                           ( t :=1020,  o := 1),   // evening 21:00
                           ( t :=1440,  o := 1)    // 24:0;
                   ]));
      OUT       : NH_POI_DAYWRK ;                  // Out
      HOL       : NH_POI_DAYWRK ;                  // Holiday
   END_STRUCT;

   NH_POI_HETWRK {HIDDEN} : NH_POI := ( cx := ( p:= [       // HET  Jeden pracovny den
                           ( t :=   0,  o := 1),   // utlm     0:00
                           ( t := 360,  o := 3),   // komfort  6:00
                           ( t := 450,  o := 1),   // utlm     7:30
                           ( t := 960,  o := 3),   // komfort 16:00
                           ( t :=1380,  o := 1),   // utlm    22:30;
                           ( t :=1440,  o := 1)    // utlm    24:00;
                   ]));
   NH_POI_HETFRE {HIDDEN} : NH_POI := ( cx := ( p:= [       // HET  volny den
                           ( t :=   0,  o := 1),   // utlm     0:00
                           ( t := 420,  o := 3),   // komfort  7:00
                           ( t :=1380,  o := 1),   // utlm    23:00
                           ( t :=1440,  o := 1)    // utlm    24:00;
                   ]));
  	NH_POI_WHET  {HIDDEN} :  STRUCT
      PON       : NH_POI_HETWRK ;                  // pondelok
      UTO       : NH_POI_HETWRK ;
      STR       : NH_POI_HETWRK ;
      STV       : NH_POI_HETWRK ;
      PIA       : NH_POI_HETWRK ;
      SOB       : NH_POI_HETFRE ;
      NED       : NH_POI_HETFRE ;
      FRE       : NH_POI_HETFRE ;
      ALL       : NH_POI_HETFRE ;
      OUT       : NH_POI   := ( cx := ( p:= [
                           ( t :=   0,  o := 1),   // utlm     0:00
                           ( t :=1440,  o := 1)    // utlm    24:00;
                   ]));
      HOL       : NH_POI   := ( cx := ( p:= [
                           ( t :=   0,  o := 0),   // protimraz    0:00
                           ( t :=1440,  o := 0)    // protimraz    24:00;
                   ]));
   END_STRUCT;

   NH_POI_VENWRK {HIDDEN} : NH_POI := ( cx := ( p:= [       // HEV  Jeden pracovny den
                           ( t :=   0,  o := 0),   //
                           ( t := 300,  o := 3),   // 5:00
                           ( t := 315,  o := 0),   // 5:15
                           ( t := 720,  o := 3),   // 12:00
                           ( t := 735,  o := 0),   // 12:15
                           ( t :=1080,  o := 3),   // 18:00
                           ( t :=1095,  o := 0),   // 18:15
                           ( t :=1440,  o := 0)    //    24:00;
                   ]));

  	NH_POI_WVEN {HIDDEN} :  STRUCT
      PON       : NH_POI_VENWRK ;                  // pondelok
      UTO       : NH_POI_VENWRK ;
      STR       : NH_POI_VENWRK ;
      STV       : NH_POI_VENWRK ;
      PIA       : NH_POI_VENWRK ;
      SOB       : NH_POI_VENWRK ;
      NED       : NH_POI_VENWRK ;
      FRE       : NH_POI_VENWRK ;
      ALL       : NH_POI_VENWRK ;
      OUT       : NH_POI_VENWRK ;
      HOL       : NH_POI_VENWRK ;

   END_STRUCT;

  	NH_FRM_249  {HIDDEN} :  STRUCT          // sablona typovych dni
      hed   : NH_FRM_HED := (Name:='_249',row:=1,desc:='Typove dni');
      DAY   : NH_POI_WDAY;             // DAY   : PO-NE
      HET   : NH_POI_WHET;             // HET   : PO-NE
      VEN   : NH_POI_WVEN;             // VEN   : PO-NE
   END_STRUCT;

   NH_FRM_247	{HIDDEN}   : STRUCT
      hed      : NH_FRM_HED := (Name:='_247',wht:=0,row:=2,desc:='Typ.Day+Time slider');
      txt   : ARRAY[0..2] OF INT := [555,223,223]; 										// texty v hlavicke - riadok 1
      poi   : ARRAY[0..3] OF NH_POD_CFG :=
                              [  (),                                            // DayMode sa preberie ako default
                                 (  tim := false,  typ := 1,  n := 7,  o := 3,  // HetMode sa zadefinuje
                                     vo := ( o := [
                                                      ( o := 171,  c := 4),      // 0 - vlocka
                                                      ( o := 173,  c := 8),      // 1
                                                      ( o := 175,  c := 6),      // 2
                                                      ( o := 177,  c := 7)]),    // 3
                                   ),
                                 (  tim := false,  typ := 2,  n := 7,  o := 3,  // VEN sa zadefinuje
                                     vo := ( o := [
                                                      ( o :=  54,  c := 4),      // 0 - off
                                                      ( o := 173,  c := 8),      // 1
                                                      ( o := 175,  c := 6),      // 2
                                                      ( o := 177,  c := 7)]),    // 3
                                    ),

                                 (  tim := false,  typ := 3,  n := 4,  o := 3,  // hyst REG
                                     vo := ( o := [
                                                      ( o :=  54,  c := 4),      // 0 - off
                                                      ( o := 173,  c := 8),      // 1
                                                      ( o := 175,  c := 6),      // 2
                                                      ( o := 177,  c := 7)]),    // 3
                                    )

                               ];

   	ini 	: NH_FRM_249;
   END_STRUCT

   NH_FRM_260_DATA	{HIDDEN} : STRUCT
		mWsb		: USINT;
		typ		: SINT := -1;
		cf			: NH_OBJ_123_CF;
		txt		: NH_PI14;
		pvCmd    : NH_PV18;				//click 1-5, P,H  [switch,0,0,0,0,Push,Hold,0]
	END_STRUCT

   NH_FRM_260	 : STRUCT
      hed : NH_FRM_HED := (Name:='_260',desc:='Prepincie menu');
		grp		: USINT;				// skupina do ktorej DEV patri
		typ		: SINT := 0;      // pripadny konkretny typ DEV
		i			: USINT;
		m			: USINT;
		nWsb		: USINT := 20;   	// max pocet predvolieb
		mWsb		: ARRAY[0..20] OF NH_FRM_260_DATA := [
						( mWsb := 0,  	cf := (rw2 := 4,x:=180,y:=500),
												txt := [80,81,616,83], 									// 0 default SVD,ZAS : Nic/prepnut/zapnut/vypnut
//												cmd := [ 0, 2, 11,10]),									// cisla prikazov
												//Click  1  2  3  4  5 Pr Hl xx
											 pvCmd := [ 2, 0, 0, 0, 0, 0, 0, 0]),									// predvolba do pWsb.cmd[click1,2,3,4,5,Push,Hold,rezerva]

						( mWsb := 4, typ:=1,  	cf:= (rw2:= 8),
												txt := [80,626,625,179,182,188,189,178],     	// ROL				Nic/Start*Stop/Natacat Lamly/Vytiahnut Hore/Zatihmut dolu/Lamely otvorit/Lam.Zatvorit/Predvolba
//												cmd := [ 0,23,  24, 10, 11, 26, 27, 14]),
												//Click  1  2  3  4  5 Pr Hl xx
											 pvCmd := [23,10,11,26,27,24, 0, 0]),
						( mWsb := 4, typ:=2,  cf:=(rw2 := 7),
												txt := [80,181,618,619,183,178,72],  				// GAT{0=garaz,1=brana}		Nic/Start-stop/OtvoritZatvorit/Stop/Predvolba/Potvrdit zatvorene
//												cmd := [ 0,  2, 11, 10,  3, 14,51])
											 pvCmd := [ 2, 0, 0, 0, 0,51, 0, 0]),									// predvolba do pWsb.cmd[click1,2,3,4,5,Push,Hold,rezerva]
						( mWsb := 4,  	cf:= (rw2:= 6),
												txt := [80,81,82,159,83,84],			  				// SCN     Nic/prepnut/PV/Zapnut(100)/vypnut/stmievat
//												cmd := [ 0, 2,14, 11,10, 6]),
											 pvCmd := [ 2,11,10,14, 0, 6, 0, 0]),

						( mWsb := 5, typ:=1,  	cf:= (rw2:= 7),
												txt := [80,178,179,182,188,189,183],     	// ROL				Nic/Predvolba/Vytiahnut Hore/Zatiahmut dolu/Lamely otvorit/Lam.Zatvorit/Stop
//												cmd := [ 0,14, 10, 11, 26, 27, 3]),
												//Click  1  2  3  4  5 Pr Hl xx
											 pvCmd := [14,10,11,26,27, 3, 0]),
						( mWsb := 5, typ:=2,  cf:=(rw2 := 7),
												txt := [80,181,618,619,183,178,72],  				// GAT{0=garaz,1=brana}		Nic/Start-stop/OtvoritZatvorit/Stop/Predvolba/Potvrdit zatvorene
//												cmd := [ 0,  2, 11, 10,  3, 14,51])
											 pvCmd := [ 2, 0, 0, 0, 0,51, 0, 0]),									// predvolba do pWsb.cmd[click1,2,3,4,5,Push,Hold,rezerva]
						( mWsb := 5,  	cf:= (rw2:= 4,x:=110),
												txt := [80,118,159,83],				  					// ACT        	  	Nic/vykonat akciu/Zapnut(100)/vypnut
//												cmd := [ 0, 14, 11,10]),
											 pvCmd := [14, 0, 0, 0, 0, 0, 0, 0]),
						( mWsb := 6,  	cf:= (rw2:= 6,x:=140),
												txt := [80,154,155,156,157,223],						// HET        	  	Nic/off/1/2/3/Auto
//											  Cmd := [ 0, 31, 32, 33, 34, 30]),
											 pvCmd := [32,33,34,31, 0,30, 0, 0]),
						( mWsb :=11,  	cf:= (rw2:= 6),
												txt := [80,81,82,159,83,84],							// SVA,RGB        Nic/Prepnut/zapnut(PV)/Zapnut(100)/vypnut/stmievat
//												cmd := [ 0, 2,14, 11,10, 6]),
												//Click  1  2  3  4  5 Pr Hl xx
											 pvCmd := [ 2, 0, 0, 0, 0, 6, 0, 0]),									// predvolba do pWsb.cmd[click1,2,3,4,5,Push,Hold,rezerva]
						( mWsb :=31,  	cf:= (rw2:= 9),
												txt := [80,181,180,179,182,188,189,178,183],     	// ROL				Nic/Start*Stop/Natacat Lamly/Vytiahnut Hore/Zatihmut dolu/Lamely otvorit/Lam.Zatvorit/Predvolba
//												cmd := [ 0, 2, 25, 10, 11, 26, 27, 14, 3]),
												//Click  1  2  3  4  5 Pr Hl xx
											 pvCmd := [ 2,10,11,26,27,25, 3, 0]),

						// ak ma skupina viac typov, prve musia byt najs konkretne typy, a za za nimi na koniec -1
						( mWsb :=37, typ:=2,cf:=(rw2:=3),
												txt := [80,617,72],      								// GAT{dvere}		Nic/Otvorit/Potvrdit zatvorene
//												cmd := [ 0, 2, 51]),
											 pvCmd := [ 2, 0, 0, 0, 0,51, 0, 0]),									// predvolba do pWsb.cmd[click1,2,3,4,5,Push,Hold,rezerva]
						( mWsb :=37, typ:=3,  cf := (rw2 := 3),
												txt := [80,617,72],      								// GAT{branicka}	Nic/Otvorit/Potvrdit zatvorene
//												cmd := [ 0, 2, 51]),
											 pvCmd := [ 2, 0, 0, 0, 0,51, 0, 0]),									// predvolba do pWsb.cmd[click1,2,3,4,5,Push,Hold,rezerva]
						( mWsb :=37,  cf:=(rw2 := 7),
												txt := [80,181,618,619,183,178,72],  				// GAT{0=garaz,1=brana}		Nic/Start-stop/OtvoritZatvorit/Stop/Predvolba/Potvrdit zatvorene
//												cmd := [ 0,  2, 11, 10,  3, 14,51])
											 pvCmd := [ 2, 0, 0, 0, 0,51, 0, 0])									// predvolba do pWsb.cmd[click1,2,3,4,5,Push,Hold,rezerva]
					];
	END_STRUCT

   NH_LOG_IMP       : STRUCT   // struktura EVN-log
		ok				: STRING[1]:=' ';  		sok	: BYTE := 16#3b;
		cf				: STRING[3];   			s1 	: BYTE := 16#3b;
      cfg         : STRING[3];     			s2 	: BYTE := 16#3b;
      ID          : STRING[5];   			s6 	: BYTE := 16#3b;         // nacitane z exportu
  		inv			: string[1]:='0';      	s3i 	: BYTE := 16#3b;			 // on/off
  		typ			: string[1]:='0';      	s3 	: BYTE := 16#3b;
  		typYes		: string[1]:='N';      	sy 	: BYTE := 16#3b;				// prepisuje sa typ
		d				: STRING[1]:='0';			d2 	: BYTE := 16#3b; 				//	hw.d[d]
      HWs         : STRING[8];      		sa 	: BYTE := 16#3b;
		HWtyp			: STRING[1]:= '0';		d22 	: BYTE := 16#3b;
      IO          : STRING[1];      sb 	: BYTE := 16#3b;         // I=vstup, Q=vystup, M=pamat
      MEM         : STRING[1];      sc 	: BYTE := 16#3b;         // 0=BOOL,1=REAL,
      RomID       : STRING[3]:='   ';     s7 	: BYTE := 16#3b;         // RomID, ktore sa bude hladat v xRom^.cf.ID
      Rom         : STRING[3]:='   ';     s5 	: BYTE := 16#3b;         // cislo vety rom {nd}
      typRom      : STRING[1]:=' ';    	s4 	: BYTE := 16#3b;			 // 0=admin,1=vnutorna,2=vonkajsia,3=podzemna,4=wellmess,5=sauna
      Name        : STRING[20];     s8 	: BYTE := 16#3b;
      NameCf      : STRING[20];     s81 	: BYTE := 16#3b;          		// aktualny nazov v CFG
      Cr       	: BYTE   := 16#0D;
      Lf       	: BYTE   := 16#0A;
	END_STRUCT;

   NH_FRM_500	{HIDDEN}   : STRUCT
      hed      : NH_FRM_HED := (Name:='_500',desc:='Import from CIB');
		rImp		: NH_LOG_IMP;
		eImp 		: NH_LOG_IMP;
   END_STRUCT

	NH_brw_D1_BLK    {HIDDEN}  :  NH_OBJ_DAT  :=          // PIR
      (wh:=0, x:=125,  y:=109,  w:=48, h:= 68, FgC:=4,  BgC:=2,  fn:=0, cf:=(c:=0) ); // 5 Blk
	NH_brw_D1_PIR    :  NH_OBJ_DAT  :=          // PIR
      (wh:=0, x:=125,  y:=109,  w:=50, h:=68 , FgC:=7,  BgC:=2,  fn:=0, cf:=(c:=5)); // 6 PIR day mode

	NH_OBJ_LIST   :  NH_OBJ_DAT  :=          // obrazok dev list
      (wh:=1, x:=x2-110,y:=109,w:=48, fn:=39, cm:=80); // 6 list DEV

	NH_brw_OBJ  {HIDDEN}   :  STRUCT
		list		: NH_OBJ_LIST;
		dlgl		: NH_OBJ_LIST := (fn:=333);
		rgbwa		: NH_OBJ_DAT  := (wh:=20, x:=125,  y:=109,  w:=50, h:=60 , FgC:=11,  BgC:=2,  fn:=0, cf:=(c:=4,n:=0,p:=0)); // 5 RGBWA na sebe
		srgbwa	: NH_OBJ_DAT  := (wh:=20, x:=x2-110,  y:=109,  w:=50, h:=0 ,  FgC:=11,  BgC:=2,  fn:=0, cf:=(c:=5,n:=0,p:=0)); // 6 RGBWA na sebe
//		srgbwa	: NH_OBJ_DAT  := (wh:=20, x:=125,  y:=109,  w:=50, h:=0 ,  FgC:=10,  BgC:=2,  fn:=0, cf:=(c:=4,n:=0,p:=0)); // 6 RGBWA na sebe
		blk		: NH_BRW_D1_BLK := (wh:=20);
//		tim_1    : NH_OBJ_4O1 := (wh:=107,obj:=2,ok:=[0,1,0,0],obr:=[0,295,0,0]); 		// timer nad hlavnym obrazkom, def
//		tim_2    : NH_OBJ_4O2;
	END_STRUCT

END_TYPE

TYPE

   NH_LIST_OBR	     :  STRUCT

      ok       : ARRAY[0..1]      OF INT := [35,38];                                                                  // 0/1
      ko       : ARRAY[0..1]      OF INT := [38,35];                                                                  // 1/0
		man		: ARRAY[0..1]      OF INT := [220,221];                                                                // manual = ruka
      day      : ARRAY[0..1,0..4] OF INT := [139,141,143,145, 66, 140,142,144,146, 69 ];                              // Day/Evening/Night/Morning/Lock
      day2  	: ARRAY[0..1,0..3] OF INT := [139,141,143,145,
															140,142,144,146];                              // Day/Evening/Night/Morning
      Lck2  	: ARRAY[0..1,0..3] OF INT := [ 66,389,130,131,
															388,390,391,392];                              // Unlock/Lock/Dark/Light

//      RGB      : ARRAY[0..1,0..4] OF USINT := [208,208,208,208,208, 208,210,209,212,211 ];                              // w-R-G-B-orange
      RGB      : ARRAY[0..4] OF INT := [208,210,209,212,211 ];                              // w-R-G-B-orange
      RGBWA    : ARRAY[0..1,0..5] OF INT := [208,208,208,208,208,208,   208,210,209,212,371,211 ];                              // w-R-G-B-orange
      led      : ARRAY[0..1,0..7] OF INT := [208,208,208,208,208,208,208,208,  209,210,209,210,209,210,209,210];      // Green/Red
      ledR     : ARRAY[0..1,0..1] OF INT := [208,208,  210,209];                                                      // Red/Green - ked je prva RED
      off      : ARRAY[0..1]      OF INT := [127,128];                                                                // Zablokovat 0/1
      Dark     : ARRAY[0..1]      OF INT := [130,131];                                                                // Dark
      pir      : ARRAY[0..1,0..5] OF INT := [139,141,143,145,067,130, 140,142,144,146,069,131 ];                        // Day/Evening/Night/Morning/0/Twilight

      clrh     : ARRAY[0..4]      OF INT := [4,8,6,7,2];                                                              // siva/zelena/oranzova,cervena
      OFFon    : ARRAY[0..1]      OF INT   := [54,400];                                                                 // OFF=siva off, ON = zeleny podklad ON
      run      : ARRAY[0..1]      OF INT := [226,227];                                                                // RUN off/ON
//      LedGBR   : ARRAY[0..2,0..4] OF USINT := [139,141,143,145, 66, 140,142,144,146, 69 ];                              // Day/Evening/Night/Morning/Lock

   END_STRUCT;

   NH_TYPE_MNU	      :  STRUCT 		               // definicia spodneho menu
      x        : ARRAY [1..6,3..8] OF INT :=                 // [pocet menu , suradnice ciala menu[3,4,5,6,7,8] ]
                        [           xc,          0,          0,          0,          0,             0,    // 1 x Mnu
                               xc-xz/2,    xc+xz/2,          0,          0,          0,             0,    // 2 x Mnu
                                 xc-xz,         xc,      xc+xz,          0,          0,             0,    // 3x menu
                            xc-xz/2-xz,    xc-xz/2,    xc+xz/2, xc+xz/2+xz,          0,             0,    // 4x menu
                               xc-xz*2,       xc-xz,        xc,      xc+xz,    xc+xz*2,             0,    // 5x menu (HOME)
                          xc-xz*2-xz/2,  xc-xz-xz/2,   xc-xz/2,    xc+xz/2, xc+xz+xz/2,  xc+xz*2+xz/2     // 6x menu (zakladne)
                         ];

      m        : ARRAY [0..31,0..2] OF INT :=              // [[typ menu], [fn,wh,cm]
                        [  0,  0,  0,                        //  0- nic
                          23, 24,  3,                        //  1-setup   DEV
                         120,121,  1,                        //  2-Casove udaje (oneskorene zapnutie/vypnutie, max.cas zapnutia)
                         122,123,  2,                        //  3-LEVEL
                          83, 84,121,                        //  4-tune LED predradnik
                         196,197,  7,                        //  5-Blikanie
                         121,125,  4,                        //  6-RGB-COLOR

                          61, 61, 10,                        //  7-HET/pv-TVE - teploty s obrazkom teploty
                         190,191, 12,                        //  8-HET     - rozdiely teplot pre kurenie
                         345,345, 11,                        //  9-TVE/KOT - uroven otvorenia ventilu
                         220,221, 13,                        // 10-HET/TVE/KOT - rucne
                         222,223, 14,                        // 11-HET - automatika (casove plany)
                          23, 24, 15,                        // 12-TVE - setup = typ ventilu
                          83, 84, 16,                        // 13-TVE - tune = parametre + tools + adaptacia/kalibracia
                         224,225, 20,                        // 14-TVE - tools / adaptacia + kalibracia
                         273,274,199,                        // 15-DaofWeek - nastavenie typu aktualneho dna

                         261,262, 31,                        // 16-ROL-veterna automatika
                         110,111, 32,                        // 17-ROL-kalibracia
                          83, 84, 33,                        // 18-ROL-pozicie/castune
                          23, 24, 34,                        // 19-ROL-setup
                         139,148, 35,                        // 20-ROL-vychod slnka

                          33, 34,  5,                        // 21-WSB play/Led/Setup
                         204,205,120,                        // 22-WSB-Led
                          23, 24,  6,                        // 23-WSB-setup
                          23, 24, 40,                        // 24-BRA-setup

                          83, 84, 23,                         // 25-VEN-tune
                         120,121,198,                         // 26-Systemovy cas, datum ...
                         311,311,122,                         // 27-TGL-Display - svietivost
                         311,311,123,                         // 28-TGL-display - nastavit co sa zobrazuje
                         345,345, 10,                         // 29 HET teploty s obrazkom predvolby
                          83, 84, 21,                        // 30 HET/TVE - regulacne odozvy teploty
                         348,348, 82                         // 31 priradit do ROM

                          ];

 	END_STRUCT;

END_TYPE

VAR_GLOBAL
	xObrWht						{HIDDEN}	: PTR_TO NH_OBR_WHT;
   yFrmName AT mObr  		{HIDDEN} : NH_FRM_HED;              // head of template
	yFrmData	AT mObr[34]		{HIDDEN} : USINT;	//NH_LOG_HEAD;		// data of template
	yFrm_229	AT	mObr			{HIDDEN}	: NH_FRM_229;	// obrazky predvolieb regulatorov
	yFrm_230	AT	mObr			{HIDDEN}	: NH_FRM_230;	// obrazky DEV
	yFrm_231	AT	mObr			{HIDDEN}	: NH_FRM_231;	// obrazky pre stav DEV,CAT,...
	yFrm_232	AT	mObr			{HIDDEN}	: NH_FRM_232;	// obrazky HOM,CAT
	yFrm_233	AT	mObr			{HIDDEN}	: NH_FRM_233;	// xObs
	yFrm_234	AT	mObr			{HIDDEN}	: NH_FRM_234;	// xFiD
	yFrm_235	AT	mObr			{HIDDEN}	: NH_FRM_235;
	yFrm_236	AT	mObr			{HIDDEN}	: NH_FRM_236;
	yFrm_246	AT	mObr			{HIDDEN}	: NH_FRM_246;
	yFrm_247	AT	mObr			{HIDDEN}	: NH_FRM_247;
	yFrm_260	AT mObr			{HIDDEN} : NH_FRM_260;
	yFrm_248	AT	mObr			{HIDDEN}	: NH_FRM_248;

(*
	yFrm_011		AT	mObr	{HIDDEN}		: NH_HOM_011;	// HOM
		yFrm_030		AT	mObr	{HIDDEN}		: NH_FRM_030;	// AUT-MAN
	yFrm_039		AT	mObr	{HIDDEN}		: NH_FRM_039;	// FRM-TGL-LED
		yFrm_076		AT	mObr	{HIDDEN}		: NH_FRM_076;	// AUT-MAN

//	yFrm_230		AT	mObr	{HIDDEN}		: NH_FRM_230;	// obrazky DEV

	yFrm_247		AT	mObr	{HIDDEN}		: NH_FRM_247;

*)

	// na ladenie
(*
	yFrm_061		AT mObr	{HIDDEN} 	: NH_FRM_061;
	yFrm_260		AT mObr	{HIDDEN} 	: NH_FRM_260;
	yFrm_005		AT mObr	{HIDDEN} 	: NH_FRM_005;
	yFrm_001		AT mObr	{HIDDEN} 	: NH_FRM_001;					// HW par DLI
	yFrm_091		AT mObr	{HIDDEN} 	: NH_FRM_091;					// HW par DLI
*)
END_VAR

TYPE

   NH_WEB_SS	{HIDDEN}  : STRUCT
      newLogin : BOOL;
   END_STRUCT
   NH_WEB_PD	{HIDDEN}  : STRUCT
      usr      : USINT;          // prihlaseny user na stranke
      new      : BOOL;
      usage    : USINT;
   END_STRUCT
   NH_WEB_IP	{HIDDEN}  : STRUCT
      pg      : USINT;          // prihlaseny user na stranke
      ip      : TIPadr;
      new     : BOOL;
   END_STRUCT
   NH_WEB_PG	{HIDDEN}  : STRUCT
      pg      : ARRAY [1.._Nh_WEB_M] OF NH_WEB_PD;       // stav usrov
      ip      : ARRAY [1..8] OF NH_WEB_IP;             // novo prihlasena IP
      ses     : USINT;                                // pocet aktivnych session
   END_STRUCT

   NH_WEB_ACC 	{HIDDEN} : STRUCT
      wO 	   : TWebServerAccessTable;   	          // Old web acces table
      wA 	   : TWebServerAccessTable;   	          // NEW web acces table
      pgN      : NH_WEB_PG;
      pgO      : NH_WEB_PG;
      WebChg   : UINT;
   END_STRUCT

  	NH_SLD_POX {HIDDEN} :  STRUCT     // struktura pre slider z viacerych casovych pointov
      mx       : REAL;
      my       : REAL;
      xy       : ARRAY[0..1,0..7] OF INT;             // suradnica zobrazeneho casu nad vynasacou ciarou pointu 0=x,1=y
  	END_STRUCT;

  	NH_SLD_CPY  {HIDDEN}  :  STRUCT     // struktura pre slider z viacerych casovych pointov
      all      : BOOL;                                // je vybraty zdrojovy den pre kopirovanie, nemenia sa dni, len sa oznacuju do kopirovania
		chk		: BOOL;											// aspon jeden DEV je oznaceny na cpy
      cpy      : BOOL;                                // je vybraty zdrojovy den pre kopirovanie, nemenia sa dni, len sa oznacuju do kopirovania
		src		: USINT;											// zdrojovy den
		dst		: NH_BTN15;                            // ciele kam sa bude kopirovat
  	END_STRUCT;

  	NH_OBJ_DSH {HIDDEN} :  STRUCT       // velkost: 30  vseobecny objekt
      wh       : USINT := 102;                  // 0=nic,1=obrazok...2=...
		x			: INT ;                     		// 1 x-ova suradnica stredu objektu
		y			: INT ;         				      // 3 y-ova suradnica stredu objektu (default pre spodne menu)
		w			: INT := 80;            		   // 5 sirka  (pri obrazku je to aj vyska)
      cm       : USINT := 251;                  // 11 command, ktory vrati pri stlaceni
		dash		: INT			:= 381;      			// 7	cislo obrazkaDSH
		vMin		: REAL		:= 0.0;					// 9  minimalna hodnota
		vMax		: REAL		:= 18.0;					//	13 max.hodnota pre zobrazenie
		tx1		: STRING[3] := 'Min';				// 17 text laveho intervalu : Min,Avg, pravy je vzdy Max
		title		: INT;									// 21 cislo textu dash
		idx		: USINT;                         // 23 index na aMeteo.idx[]
//		tx2		: STRING[3] := 'Max';            // 21
		mj			: STRING[3]; 							// 25	popis jednotky °C, %, hPa

      Qr       : BOOL;                            // 29 zaciatok dotyku (tch = true )
      Qf       : BOOL;                            // koniec dotyku (tch = true )
      Qs       : BOOL;                            // koniec dotyku slidera
      btn      : BOOL;                            // univerzalne pouzitelny btn
      kxy      : BOOL;                            // priznak, ze uz bolavykonana korekcia xy suradnice
      nTch     : BOOL;                            // tento obj sa len zobrazuje,necaka sa dotyk
      prs      : BOOL;                            // nad tymto objektom je povoleny press
      tch      : BOOL;                             // dotyk/press bol na tomto objekte

	END_STRUCT;                      					// 30 byte

  	NH_OBJ_124   {HIDDEN}   :  STRUCT    // prepinac medzi obrazkami, alebo chck 15 obrazkov v 2 riadkoch
      // prvy riadok
      wh       : USINT 	:= 124;
		x			: INT 	:= 60;                  	// x-ova suradnica stredu objektu 1.obrazka
		y			: INT 	:= y1+130;         			// y-ova suradnica stredu objektu 1.obrazka
      w        : INT 	:= 490;                    // velkost obrazka
      cm       : USINT 	:= 251;                  	// ... len pre kompatilititu
      h        : INT 	:= 50;                     // vzdialenost medzi obrazkami
		nObr		: USINT	:= 7;								// pocet obrazkov
		Obr1 		: USINT	:= 1;                      // cislo prveho obrazka
      aVar  	: UDINT;                           	// adresa cielovej premennej, kde sa uklada posledny vyber
      typ      : USINT 	:= 1;                     	// typ cielovej premennej 1=usint,3=sint
      aArray	: UDINT;                           	// adresa cieloveho pola
		WrkVar	: USINT;										// pomocna premenna - ak sa cislo vyberu neuklada do nejakej premennej je va adrese aVar tato premmenne,
		WrkArray	: NH_BTN15;									// pomocne pole [0..15]
      FgC      : USINT 	:= 4;                     	// oramovanie vybrateho riadka = kruznica
      BgC      : USINT 	:= 4;                     	// vypln kruznice
		// 27
		xxxx     : INT 	:= 28;                           // vyska textu
      // bit 29
		Visible	: BOOL := true;							// len zobrazit
		Enable	: BOOL := true;							// povolenie vyberat
		Chceck	: BOOL := true;                    	// vybera vsetky volby (ink len jednu a ostatne nuluje)
		Circle	: BOOL := true;							// oramovanie vyberu je kruznica
		Set4		: BOOL;                             //
		Set5		: BOOL;
		set6		: BOOL;
      Q        : BOOL;									  // xA^.trg.Q - musi si nulovat objekt
		// bit 30
      Qr       : BOOL;                            // xA^.trg.Qr
		Qf       : BOOL;                            // xA^.trg.Qf
      Qs       : BOOL;                            // toto pouziva objekt, nenastavuje sa nikde - koniec dotyku slidera, ....
      btn      : BOOL;                            // univerzalne pouzitelny btn
      kxy      : BOOL;                            // priznak, ze uz bolavykonana korekcia xy suradnice
      nTch     : BOOL;                            // tento obj sa len zobrazuje,necaka sa dotyk
      prs      : BOOL;                            // nad tymto objektom je povoleny press
      tch      : BOOL;                             // dotyk/press bol na tomto objekte

      // druhy riadok
		xTxt		: INT 	:= 60;                  	// x-ova suradnica stredu objektu 1.obrazka
		yTxt		: INT 	:= y1+130;         			// y-ova suradnica stredu objektu 1.obrazka
      wTxt     : INT 	:= 490;                    // velkost obrazka
      hTxt     : INT 	:= 25;                     // vzdialenost medzi obrazkami
      FgTxt    : USINT 	:= 2;                     	//

		ObrOff      : ARRAY[1..8] OF INT :=        	// nevybraty obrazok obrazka
							[120,148,147,130,131,378, 33];   	// nacasovat/SunRise/SunSet/DarkOff/DarkOn/random/odpocita cas od spustenia
      ObrSet      : ARRAY[1..8] OF INT :=          // vybraty obrazok
							[121,148,147,130,131,378, 34];
      TxtSet      : ARRAY[1..8] OF INT :=          // cislo textu k vybratemu obj
							[543,544,545,546,547,548,549];
		CmdSet      : ARRAY[1..8] OF USINT;          // doplnujuci CMD co sa ma urobit po vybere, normalne nic
		Dummy9		: ARRAY[1..25] OF USINT;
		// koniec 4.riadka
	END_STRUCT;

  	NH_OBJ_ROL  {HIDDEN} :  STRUCT       // velkost: 30  ROLETY zobrazenie
      wh       : USINT 	:= 109;         			// 0
		x			: INT		:= 50;                  // 	lavy horny roh ROL -
		y			: INT 	:= 200;                 //
		w			: INT 	:= 430;			         // 	sirka ROL
		cm			: USINT  := 251;                 // 7	len pre kompatibilitu
		h			: INT 	:= 658;			         // 	vyska ROL
		// 11
		yCirRol	: INT;                 				// 	suradnica gulicky ROL
		yCirLam	: INT; 			         			// 	suradnivc gulicky LAM

		bRol     : INT		:= 50;	                  // 10	vyska boxu nad roletou
		xLam		: INT		:= 530;                 // 	lavy horny roh LAM slidera
		yLam		: INT 	:= 220;
		xObrR		: INT		:= 80;                  // 	x-suradnica obrazka rolety
		wObr		: USINT	:= 60;						//	 	sirka/vyska obrazku
			cf			: NH_DEV_IO;							//23	 byte 23
      // byte 29
		dummy0	: BOOL;                          // byte 29
		dummy1	: BOOL;
		dummy2	: BOOL;
		dummy3	: BOOL;
		dummy4	: BOOL;
wwwWindGuardOn	: BOOL;                            // bezi ochrana pred vetrom
wwwHandBlkWind	: BOOL;							  	  // priznak rucneho blokovania WindG
      Q        : BOOL;									  // xA^.trg.Q - musi si nulovat objekt
		// byte 30
      Qr       : BOOL;                            // xA^.trg.Qr
		Qf       : BOOL;                            // xA^.trg.Qf
      Qs       : BOOL;                            // toto pouziva objekt, nenastavuje sa nikde - koniec dotyku slidera, ....
      btn      : BOOL;                            // univerzalne pouzitelny btn
      kxy      : BOOL;                            // priznak, ze uz bolavykonana korekcia xy suradnice
      nTch     : BOOL;                            // tento obj sa len zobrazuje,necaka sa dotyk
      prs      : BOOL := true;                    // nad tymto objektom je povoleny press
      tch      : BOOL;                             // dotyk/press bol na tomto objekte

		// obj 2 = 30 byte (0 byte )
      wh2      : USINT 	:= 0;  							//0	wh v 2 objekte
		rCirSld	: INT		:= 30;							// 	r gulicky slidera
		rCirUpDn	: INT		:= 35;							// 	r gulicky slidera	pri zobrazeni pohyby
		wObrInfo	: INT		:= 90;							// 	velkost info obrazka
		corner	: INT 	:= 3;

wwwCMD		: USINT;										// 	co sa ma urobit
			wwwCMDf		: USINT;										//
		wSldLam	: INT 	:= 14;							//	 	hrubka aktivnej casi slidera

		hLam		: INT 	:= 615;		            // 	vyska * dlzka slidera odhora nadol
		xObrL		: INT		:= 335;	                  // 	x-suradnica obrazka LAM
		yObr		: INT		:= 900; 						// 	y-suradnica obrazkov a textu % pod  Rol

		hTxt		: USINT	:= 34;							// 	vyska textu
wwwpRol		: USINT;										// 	poziadavka na ROL v %
wwwpLam		: USINT;										// 	poziadavka na LAM v %
		// 19
		nLam		: USINT 	:= 16;							// 	pocet lamiel
		wLMax   	: INT 	:= 40;                     // 	sirka {vyska} lamely pri uplnom zaklopeni
		wLold		: INT 	:= 40;							// 	minimalna vyska lamely pri uplnom otvoreni
		mLam		: INT 	:= 10;							// 	bocny okraj medzi lamelou a lavym/pravym oranovanim
      chk    	: BOOL;                             // 28 .. odpoveda Qr
		SldRol	: BOOL := true;							// 	zobrazit slider ROL   .. odpoveda Qf
		SldLam	: BOOL := true;							// 	zobrazit slider LAM
		tchLam	: BOOL := true;							// 	povolit nastavovanie slidera LAM
		tchUpDn	: BOOL := 0;								// 	pri dotyku len spustit zmenu smeru  CMD=1 .. ma prednost pre sliderom ROL
		StatRow	: BOOL := true;							// 	vykresluju sa aj statusove obrazky a hodnoty pod obrazkom
		ShwLamUp	: BOOL := true;							// 	vykresluju sa aj statusove obrazky a hodnoty pod obrazkom
	END_STRUCT;                      					// 60 byte

  	NH_ROW {HIDDEN} :  STRUCT              // jedne riadok
      h        : NH_ROW_H;
      o        : NH_ROW_O;
	END_STRUCT;

 	NH_FIL {HIDDEN} :  STRUCT 		          	   // hlavicka a FILTER aktualneho browsu
      cf          : NH_DEV_IO;                  // identifikacia DEV
		dev			: FILT_LIST; 		            // hlavny filter pre DEV
		cat			: FILT_LIST; 		            // hlavny filter pre CAT
      rom         : USINT;                      // filter na rom
      typ         : SINT;                       // filter na TYP
	END_STRUCT;

  	NH_TCH {HIDDEN} :  STRUCT
		aObj			: UDINT;
      evn         : USINT;                            // vyhodnotene cislo udalosti
      cmd         : USINT;                            // vysledny prikaz podla udalosti 20=home screen
      cm          : USINT;                            // command z objektu
      wh          : USINT;                            // wh z objektu riadka nad ktorym bol posledny dotyk   xR^.o.ob[0].wh
      wht         : SINT;

      cmdNext       : USINT;
      xMwht        : SINT;
      col         : SINT :=  1;                       // stlpec v riadku
      row         : SINT := -1;                       // riadok, v ktorom bolo stlacenie
      obj         : SINT := -1;                       // objekt v riadku na ktorom bol stlacenie
      tme         : UINT;                             // cas podrzania
		x1,x2,y1,y2 : INT;                              // suradnice pri prvom/poslednom stlaceni alebo od zaciatku pres
      ok          : BOOL;                             // priznak vyhodnotenia az do najblizsieho noveho dotyku
//      mnu         : BOOL;                             // nove menu
//      tob         : BOOL;                             // na nejakom objekte bol dotyk
//      prs         : BOOL;                             // je press
//      Qpr         : BOOL;                             // impulz pri prvom vyhodnoteni (aj na nevybratom objekte)
//      Qpf         : BOOL;                             // impulz pri ukonceni press     (aj na nevybratom objekte)
      Q           : BOOL;                             // priznak stlacenia nad vybratym objektom
      Qr          : BOOL;                             // impulz pri 1.stlaceni nad vybratym objektom
      Qf          : BOOL;                             // impulz pri uvolneni stlacenia nad vybratym objektom
//      Qs          : BOOL;                             // impulz LEN pre slider - aktivuje sa pri Qf a sposobi este jednu otocku, aby sa odcitali posledne zapisane data - najma pri dotyky nad sliderom
      del         : BOOL;                             // priznak vymazania riadka (row)
      cpy         : BOOL;                             // priznak kopirovania riadka (row)
//      Bl          : BOOL;
      End         : BOOL;                             // uplne ukoncenie udalosti
      mnu         : BOOL;                             // dotyk bol na menu
      sld         : BOOL;                             // pohybujeme sliderom
      p1          : BOOL;                             // priznak s ktorym pracuje  program
      p2          : BOOL;                             // priznak s ktorym pracuje  program
   END_STRUCT;

   NH_TCH_WHT {HIDDEN} : STRUCT      				// HLAVNA RIADIACA PREMENNA
      n           : USINT;
      t           : ARRAY[0..5] OF NH_TCH;
   END_STRUCT;

  	NH_R_XY {HIDDEN} :  STRUCT
      xp          : INT := 0;                                // x-posuv celej strany
      yp          : INT := y1;                               // y-posuv celej strany
	END_STRUCT;

  	NH_SLD_POD {HIDDEN} :  STRUCT     // struktura pre slider z viacerych casovych pointov
//  		edit		: BOOL;									// priznak editacie = blokuje zmenu dna typ.dni

		edit		: NH_DEV_CF;
      btn      : BOOL;                          // bol stlaceny btn na Typ_Day
      zom      : BOOL;                          // je vybraty bod a je vyvyseny
      tch      : BOOL;                          // bol tch nad tymto obewktom
      prs      : BOOL;                          // drzime objekt = pohybujeme sa
      Qf      	: BOOL;                          // pustime objekt - impulz
      idx      : BOOL;                          // preindexovat
      day      : USINT;                         // vybraty typovy den pri editacii
      tpr      : USINT;                         // pocet cyklov  vyhodnotenie press nad navesim
		WhtPoi	: USINT;									// pre HET,HEV 0..1
//      Zon      : USINT;                         // zona, s rodicovskym rozvrhom 0,1 =Home
      poi      : int;                           // cislo vety v aCfg[26]
      p        : SINT := -1;                    // pocet pouzitych pointov :                                 VYPOCITA SA
      x        : SINT := -1;                    // vybraty point pri presuvani                               pomocne pole
      cf       : NH_POD_CFG;
   END_STRUCT;

  	NH_BRW {HIDDEN} :  STRUCT 											 // m-stranka univerzalneho browsu
      r           : ARRAY[0.._RowBrw] OF NH_ROW;             // objekty browsu znamenaju jedno DEV. Ak ma iba jedne stlpec, tak vtedy je r aj riadok
      s           : ARRAY[0.._SldNbr] OF NH_SLD_DAT;
      xy          : NH_R_XY;                                 // treba urobit korekciu xy
      rw          : USINT;                                   // aktualne naplneny pocet riadkov
      ref         : BOOL;                                   // priznak refreshovania pre brw200
      kor         : BOOL;                        // priznak, ci uz boli korigovane zlozky x,y
(*
		// toto je pre kopirovanie
		cf				: NH_DEV_IO;
      po          : NH_SLD_POD;
      cp          : NH_SLD_CPY;
      px          : NH_SLD_POX;
*)
	END_STRUCT;

  	NH_POD {HIDDEN} :  STRUCT 											 // m-stranka univerzalneho browsu
		// toto je pre kopirovanie
//		cf				: NH_DEV_IO;
      po          : NH_SLD_POD;
      cp          : NH_SLD_CPY;
      px          : NH_SLD_POX;
	END_STRUCT;

 	NH_LVL  {HIDDEN} : STRUCT 		           	    // hlavicka a FILTER aktualneho browsu
      //pg          : USINT;                       // typ stranky 0=home,2=FAV,ROMS,CAT,ACT,
      obj         : USINT;                       // objekt/typ stranky podla _NhDefObj
      vaz         : USINT;                       // cislo vazieb
      Naz         : STRING[20];                  // nazov v hlavicke lelvel
      Fil         : NH_FIL;                      // fitre DEV
      rw1         : NH_DEV_IO;                  // co je v prvom riadku
      obd         : USINT;                       // cislo objektu, kde je dsh
      dsh         : USINT := 0;                  // typ dsh : 0=home page, 1-riadok,2=3x2,3=6x2,
      fdv         : USINT;                       // filter len na jedno DEV - pomozne pole pre zapamatanie aktualneho vyberu
      srt         : USINT;                       // sposob sortovania
      vis         : BOOL := true;                // visible (to co sa deje na stranke da prenasa do hardware)
      brw         : BOOL;                        // je browser, inak form
      chk         : BOOL;                        // tento browser ma namiesto FAV chck
      fvz         : BOOL;                        // filter na vazby v tomto browsesa vypisuju len priradene vazby (riadchy z chk=true) (ide sa priamo po vazbach)
      psn         : BOOL;                        // zobrazuju sa ikony k zabezpecovacke
//      lst         : BOOL;                        // setup list HET,VEN,SCL,ACL....
      blR         : BOOL;                       	// nefiltruje miestnosti - zablokuje rom aj odstrani ikonu miestosti zo spodneho menu
	END_STRUCT;

  	NH_FRM_CAT {HIDDEN} :  STRUCT 			// enimane veliciny pre ROM,ZON
      cat         : ARRAY[0.._Nh_CAT]    OF BOOL;          // status kategorie - nieco je zapnute
   END_STRUCT;

  	NH_CAN {HIDDEN} :  STRUCT 											// definicie USRA + FAV a canvas s dotykom
      usr         : USINT;                                  // prihlaseny user = cislo vety v aCfg[22]usr musi byt na zaciatku, lebo od naz sa maze browser
      sbj         : USINT := 1;                                // subjekt = cislo vety ZON  aCfg[3]
      UsrRight    : USINT;
      nIP         : USINT;                                  // cislo IP v ramci usra
      fav         : NH_DEV_IO;
      cat         : NH_FRM_CAT;
      trg         : aTrg;                                   // triger pre dotyk na CANVAS
		CatOk			: BOOL;												// uz bol urobeny zoznam cat
      hom         : BOOL;                                   // vyvolat cisty Homepage
      admin       : BOOL;
      Logout      : BOOL;                                      // priznak zobrazenia Logout
      tch         : NH_TCH;                                 // udalost od dotyky/podrzania....
      yk          : REAL := 1.0;                            // korekcia y//      can 			: TCanvasData4096;
      can 			: TCanvasData6144;

//      can 			: TCanvasData4096;
//      can 			: TCanvasData;
	END_STRUCT;

  	NH_IXB {HIDDEN} :  STRUCT 											 // definicia browsu
      ix1         : USINT;                                   // cislo indexu 1.naplnenej vety v browse bez offset
      ix2         : USINT;                                   // cislo indexu naplenenej poslednej vety ( riadku browsu = rws)
      idx         : USINT;                                   // pocet viet od ix0;
      ofs         : USINT;                                   // ofset 1.vety v poli indexov  [0...8,8][8...10,2] ... 0,8
      n           : USINT;                                   // pocet stranok (bodov navigatora)
      w           : USINT := 50;                             // rozostup medzi bodmi
      pg          : USINT;                                   // cislo aktualnej stranky
      x1          : INT;                                     // x-suradnica 1.bodu
      row         : NH_DSH_OBJ;                              // pocet riadkov a stlpcov pre browser
	END_STRUCT;
